(* IEC 61131-3 sources: elnaProjects/ElpcLogic/PomarKc7Changed/FunctionBlocks, 112 files *)

(* ---- AOAlg.st ---- *)
FUNCTION_BLOCK AOAlg

VAR_IN_OUT
	StrAlg : struct_Alg;
END_VAR

VAR
	kran6Open : struct_PhaseAlgoritm;
	kran4Close : struct_PhaseAlgoritm;
	kran3bOpen : struct_PhaseAlgoritm;
	mvOff : struct_PhaseAlgoritm;
	kran1Close : struct_PhaseAlgoritm;
	kran2Close : struct_PhaseAlgoritm;
	kran3Close : struct_PhaseAlgoritm;
	kran5Open : struct_PhaseAlgoritm;
	autoPnsOff : struct_PhaseAlgoritm;
	pnsOn : struct_PhaseAlgoritm;
	Pg_VhodLessThen300 : struct_PhaseAlgoritm;
	Pg_VyhodLessThen300 : struct_PhaseAlgoritm;
	nu1off : struct_PhaseAlgoritm;
	nu2off : struct_PhaseAlgoritm;
	AutoNU_Off : struct_PhaseAlgoritm;
	timer600 : struct_PhaseAlgoritm;
	pnsOff : struct_PhaseAlgoritm;
	Avom1Off : struct_PhaseAlgoritm;
	Avom2Off : struct_PhaseAlgoritm;
	Avom3Off : struct_PhaseAlgoritm;
	Avom4Off : struct_PhaseAlgoritm;
	autoAVOMOff : struct_PhaseAlgoritm;
	timer5 : struct_PhaseAlgoritm;
	klapan1 : struct_PhaseAlgoritm;
	klapan2 : struct_PhaseAlgoritm;
	nu_On : struct_PhaseAlgoritm;
	Start_AO_From : struct_PhaseAlgoritm;
	fb_kran6Open : fb_ph_Kran;
	fb_pnsOn : fb_ph_Switch;
	fb_kran4Close : fb_ph_Kran;
	fb_kran3bOpen : fb_ph_Kran;
	fb_mvOff : fb_ph_SectionSwitch;
	fb_kran1Close : fb_ph_Kran;
	fb_kran2Close : fb_ph_Kran;
	fb_kran3Close : fb_ph_Kran;
	fb_kran5Open : fb_ph_Kran;
	fb_autoPnsOff : fb_ph_algoritm;
	fb_Pg_VhodLessThen300 : fb_ph_CustomPhase;
	fb_Pg_VyhodLessThen300 : fb_ph_CustomPhase;
	fb_nu1Off : fb_ph_OilPump;
	fb_nu2Off : fb_ph_OilPump;
	fb_autoNuOff : fb_ph_algoritm;
	fb_timer600 : fb_ph_Timer;
	fb_pnsOff : fb_ph_Switch;
	fb_Avom1Off : fb_ph_Switch;
	fb_Avom2Off : fb_ph_Switch;
	fb_Avom3Off : fb_ph_Switch;
	fb_Avom4Off : fb_ph_Switch;
	fb_autoAVOMOff : fb_ph_algoritm;
	fb_timer5 : fb_ph_Timer;
	fb_klapan1 : fb_ph_CustomPhase;
	fb_klapan2 : fb_ph_CustomPhase;
	fb_nu_On : fb_ph_CustomPhase;
	fb_Start_AO_From : fb_ph_CustomPhase;
	_sunpackerCommand : fb_sunpackerCommand;
	_statusAi : TYPE_StatusAi;
	_Answers : TYPE_Answers;
	_statusDualInput : TYPE_statusDualInput;
	_commandDualInput : TYPE_commandDualInput;
	_DualStateImAction : TYPE_DualStateImAction;
	_PhaseAlgoritmAction : TYPE_PhaseAlgoritmAction;
	source : BYTE;
	cmd : BYTE;
	lastCmd : BYTE;
	source_for_Status : BYTE;
	cmd_for_Status : BYTE;
	command_error_for_Status : BYTE;
	resetCmdTimer : TON;
	resetCmdTimerPriznak : BOOL;
	onInit : BOOL;
	waitReset : TON;
END_VAR

VAR_EXTERNAL
	IM : ImConfig;
	algoritms : AlgoritmsConfig;
	ai : AiConfig;
	protections : ProtectionsConfig;
	ModeGpa : TYPE_ModeGpa;
	algManager : struct_AlgoritmsManager;
	AlgTimers : struct_AlgTimers;
END_VAR

VAR CONSTANT
	Ust_Pgaza : LREAL          := 0.3;
END_VAR

IF NOT onInit THEN
    fb_kran6Open(phaseNumber:=1, act:=_on);
    fb_kran4Close(phaseNumber:=2, act:=_off);
    fb_kran3bOpen(phaseNumber:=3, act:=_off);
    fb_mvOff(phaseNumber:=4, act:=_off);
    fb_kran1Close(phaseNumber:=5, act:=_off);
    fb_kran2Close(phaseNumber:=6, act:=_off);
    fb_kran3Close(phaseNumber:=7, act:=_off);
    fb_kran5Open(phaseNumber:=8, act:=_on);
    fb_autoPnsOff(phaseNumber:=9, act:=_reset, waitCompletion:=FALSE);
    fb_pnsOn(phaseNumber:=10, act:=_on);
    fb_Pg_VhodLessThen300(phaseNumber:=11);
    fb_Pg_VyhodLessThen300(phaseNumber:=12);
    fb_nu1Off(phaseNumber:=13, act:=_off);
    fb_nu2Off(phaseNumber:=14, act:=_off);
    fb_autoNuOff(phaseNumber:=15, act:=_reset, waitCompletion:=FALSE);
    fb_timer600(phaseNumber:=16, delay:=T#600S);
    fb_pnsOff(phaseNumber:=17, act:=_off);
    fb_Avom1Off(phaseNumber:=18, act:=_off);
    fb_Avom2Off(phaseNumber:=19, act:=_off);
    fb_Avom3Off(phaseNumber:=20, act:=_off);
    fb_Avom4Off(phaseNumber:=21, act:=_off);
    fb_autoAVOMOff(phaseNumber:=22, act:=_reset, waitCompletion:=FALSE);
    fb_timer5(phaseNumber:=23, delay:=T#5S);
    fb_klapan1(phaseNumber:=24);
    fb_klapan2(phaseNumber:=25);
    fb_nu_On(phaseNumber:=26);
    fb_Start_AO_From(phaseNumber:=27);
onInit:=TRUE;
END_IF;

fb_kran6Open(StrPh:=kran6Open, Im:=Im.kran6);
fb_pnsOn(StrPh:=pnsOn, Im:=Im.pns);
fb_kran4Close(StrPh:=kran4Close, Im:=Im.kran4);
fb_kran3bOpen(StrPh:=kran3bOpen, Im:=Im.kran3b);
fb_mvOff(StrPh:=mvOff, Im:=Im.mv);
fb_kran1Close(StrPh:=kran1Close, Im:=Im.kran1);
fb_kran2Close(StrPh:=kran2Close, Im:=Im.Kran2);
fb_kran3Close(StrPh:=kran3Close, Im:=Im.Kran3);
fb_kran5Open(StrPh:=kran5Open, Im:=Im.Kran5);
fb_autoPnsOff(StrPh:=autoPnsOff, alg:=algoritms.autoPns);
fb_Pg_VhodLessThen300(StrPh:=Pg_VhodLessThen300);
fb_Pg_VyhodLessThen300(StrPh:=Pg_VyhodLessThen300);
fb_nu1Off(StrPh:=nu1off, Im:=Im.nu1);
fb_nu2Off(StrPh:=nu2off, Im:=Im.nu2);
fb_autoNuOff(StrPh:=AutoNU_Off, alg:=algoritms.autoNu);
fb_timer600(StrPh:=timer600, timer:=AlgTimers.No_wait600);
fb_pnsOff(StrPh:=pnsOff, Im:=Im.pns);
fb_Avom1Off(StrPh:=Avom1Off, Im:=Im.v1_Avom);
fb_Avom2Off(StrPh:=Avom2Off, Im:=Im.v2_Avom);
fb_Avom3Off(StrPh:=Avom3Off, Im:=Im.v3_Avom);
fb_Avom4Off(StrPh:=Avom4Off, Im:=Im.v4_Avom);
fb_autoAVOMOff(StrPh:=autoAVOMOff, alg:=algoritms.AutoAvom);
fb_timer5(StrPh:=timer5, timer:=AlgTimers.No_wait5);
fb_klapan1(StrPh:=klapan1);
fb_klapan2(StrPh:=klapan2);
fb_nu_On(StrPh:=nu_On);
fb_Start_AO_From(StrPh:=Start_AO_From);

StrAlg.CanRun := StrAlg.inCanRun;
StrAlg.OpcCommandsDisabled := StrAlg.inOpcCommandsDisabled;

IF StrAlg.isRuning THEN

    IF	(*algoritms.F3.Smazka_1_2 OR*) IM.kran1.onStatus = _statusDualInput.STATUS_ON OR IM.kran1.onStatus = _statusDualInput.STATUS_TRANSITIONAL
	    OR IM.kran2.onStatus = _statusDualInput.STATUS_ON OR IM.kran2.onStatus = _statusDualInput.STATUS_TRANSITIONAL  THEN
	    IF (*(algoritms.F3.Smazka_1_2 OR*) IM.kran1.onStatus = _statusDualInput.STATUS_ON OR IM.kran1.onStatus = _statusDualInput.STATUS_TRANSITIONAL AND NOT klapan1.start AND NOT kran1Close.top THEN
		    runPhase(klapan1);
	    END_IF;
	    IF (*algoritms.F3.Smazka_1_2 OR*) IM.kran2.onStatus = _statusDualInput.STATUS_ON OR IM.kran2.onStatus = _statusDualInput.STATUS_TRANSITIONAL AND NOT klapan2.start AND NOT kran2Close.top THEN
		    runPhase(klapan2);
    	END_IF;
	(*algoritms.F3.Smazka_1_2:=FALSE; у меня нет такой штуки*)
    END_IF;

   (* IF NOT kran6Open.start THEN
	    ystavki.Block_kr6_alg.setValue (1);
	    IF IM.kran6._cmdreset.IN = FALSE THEN
		    ystavki.Block_kr6_alg.setValue (0); такой штуки тоже нет
		        runPhase(kran6Open);
	    END_IF;
    END_IF;*)

    (*IF NOT kran4Close.start THEN
	    ystavki.Block_kr4_alg.setValue (1);
	    IF IM.kran4._cmdreset.IN = FALSE THEN
		    ystavki.Block_kr4_alg.setValue (0);
		    kran4Close.run();
	    END_IF;
    END_IF;*)

    (*IF NOT kran3bOpen.start THEN
	    ystavki.Block_kr3b_alg.setValue (1);
	    IF IM.kran3b._cmdreset.IN = FALSE THEN
		    ystavki.Block_kr3b_alg.setValue (0);
		    runPhase(kran3bOpen);
	    END_IF;
    END_IF;*)

    resetDiProtection(protections.mvOff);
    resetDiProtection(protections.Off_avar_vikluchatel);
    resetDiProtection(protections.Reg_vozb_off);
    resetDiProtection(protections.Kran1_sdvig);
    resetDiProtection(protections.Kran2_sdvig);
    runPhase(mvOff);

    (*IF NOT kran1Close.start THEN
	ystavki.Block_kr1_alg.setValue (1);*)
	    (*IF IM.kran1._cmdreset.IN = FALSE THEN
		    ystavki.Block_kr1_alg.setValue (0);
		    runPhase(kran1Close);
	    END_IF;
    END_IF;*)

    (*IF NOT kran2Close.start THEN
	    ystavki.Block_kr2_alg.setValue (1);
	    IF IM.kran2._cmdreset.IN = FALSE THEN
		    ystavki.Block_kr2_alg.setValue (0);
		    runPhase(kran2Close);
	    END_IF;
    END_IF;*)

    (*IF NOT kran3Close.start THEN
	    ystavki.Block_kr3_alg.setValue (1);
	    IF	IM.kran3._cmdreset.IN = FALSE THEN
		    ystavki.Block_kr3_alg.setValue (0);
		    runPhase(kran3Close);
	    END_IF;
    END_IF;*)

    (*IF kran6Open.top THEN
	    algoritms.S_Vibr.CanRun:=FALSE;
	    algoritms.S_Vibr.reset ();
    END_IF;*)

    IF klapan1.start AND kran1Close.top THEN
	    (*IM.Kr1_Smazka.impulse();*)
	    klapan1.top:=TRUE;
    END_IF;
    IF	klapan2.start AND kran2Close.top THEN
	    (*zIM.Kr2_Smazka.impulse();*)
	    klapan2.top:=TRUE;
    END_IF;

    (*IF 	kran1Close.top AND kran2Close.top AND kran3Close.top AND kran4Close.top AND NOT kran5Open.top THEN
	    IF	NOT	kran5Open.start THEN
            ystavki.Block_kr5_alg.setValue (1);
		    IF	IM.kran5._cmdreset.IN = FALSE THEN
			    ystavki.Block_kr5_alg.setValue (0);
			    runPhase(kran5Open);
		    END_IF;
	    END_IF;

	    resetAiProtection(protections.Pgaza_na_vyhode_nagnetatelia);
    END_IF; *)

    IF mvOff.top (*AND NOT flag1*) THEN
	    (*algoritms.AutoPNS_Start.canrun :=FALSE;
	    algoritms.AutoPNS_Start.reset ();*)
	    algoritms.autoPns.canrun :=FALSE;
	    runPhase(autoPnsOff);
	    runPhase(pnsOn);
	    runPhase(nu_On);
	    (*vkluchit nasosi*)
	    algoritms.autoNu.canrun:=FALSE;
	    (*algoritms.autoNu_2.reset ();
	    algoritms.autoNu_1.canrun:=TRUE;
	    algoritms.autoNu_1.run ();
	    flag1:=TRUE;*)
    END_IF;

    IF	IM.nu1.onStatus =_statusDualInput.STATUS_ON OR IM.nu2.onStatus =_statusDualInput.STATUS_ON AND nu_On.start AND NOT nu_On.top THEN
	    nu_On.top:=TRUE;
    END_IF;

    IF kran5Open.top THEN
	    runPhase(Pg_VhodLessThen300);
	    runPhase(Pg_VyhodLessThen300);
	END_IF;

    IF Pg_VhodLessThen300.start AND NOT Pg_VhodLessThen300.top THEN
	    IF ai.Pgaza_na_vhode_nagnetatelia.interval >= _statusAi.NORMAL AND ai.Pgaza_na_vhode_nagnetatelia.value < 0.3 THEN
		    Pg_VhodLessThen300.top:=TRUE;
	    END_IF;
    END_IF;

    IF Pg_VyhodLessThen300.start AND NOT Pg_VyhodLessThen300.top THEN
	    IF ai.Pgaza_na_vyhode_nagnetatelia.interval>=_statusAi.NORMAL AND ai.Pgaza_na_vyhode_nagnetatelia.value < 0.3 THEN
		    Pg_VyhodLessThen300.top:=TRUE;
	    END_IF;
    END_IF;

    IF Pg_VhodLessThen300.top AND Pg_VyhodLessThen300.top AND pnsOn.top AND nu_On.top AND mvOff.top THEN
	    runPhase(nu1Off);
    	    resetAiProtection(protections.dPmaslo_gaz);
	    resetDiProtection(protections.dPmaslo_gaz_less100);
	    runAiProtection(protections.Pgaza_na_vhode_nagnetatelia_GPA_STOP);
	    runAiProtection(protections.Pgaza_na_vyhode_nagnetatelia_GPA_STOP);
	    AutoNU_Off.top:=TRUE;
    	(*algoritms.autoNu_1.CanRun:=FALSE;
	    algoritms.autoNu_1.reset ();*)
    END_IF;

    (*IF nuOff.top THEN
	    IF NOT algmanager.reg_V AND NOT pnsoff.start THEN
		    runPhase(timer600);
	    END_IF;
	    IF	NOT pnsoff.start THEN
		    sbrosVibeg.ask();
	    END_IF;
    END_IF;*)

    IF timer600.top (*OR sbrosVibeg.answer=Answers.ANS_YES*)  THEN
	    runPhase(pnsOff);
	    resetAiProtection(protections.Pmaslo_sm_nizkoe);
	    resetAiProtection(protections.Pmaslo_sm_vysokoe);
	    (*resetPhase(sbrosVibeg);*)
	    resetPhase(timer600);
	    (*algoritms.F2_Ch.autoAVOM_canrun_flag:=FALSE;
	    algoritms.F2_R.autoAVOM_canrun_flag:=FALSE;*)
    END_IF;

    IF (*NOT algoritms.F2_Ch.autoAVOM_canrun_flag AND NOT algoritms.F2_R.autoAVOM_canrun_flag AND*) pnsoff.start THEN
	    runPhase(Avom1Off);
	    runPhase(Avom2Off);
	    runPhase(Avom3Off);
	    runPhase(Avom4Off);
	    (*algoritms.R_AutoAVOM.CanRun:=FALSE;
	    algoritms.R_AutoAVOM.reset();
	    algoritms.S_AutoAVOM.CanRun:=FALSE;
	    algoritms.S_AutoAVOM.reset();
	    algoritms.Auto_Avom_.CanRun:=FALSE;*)
	    runPhase(autoAVOMOff);
    END_IF;

    IF pnsOff.top AND Avom1Off.top AND Avom2Off.top AND Avom3Off.top AND Avom4Off.top AND autoAVOMOff.top  THEN
	    runPhase(timer5);
    END_IF;

    IF timer5.top THEN
	    runPhase(timer5);
    END_IF;
END_IF;

_sunpackerCommand(command := StrAlg.inCommand);
	source := _sunpackerCommand.source;
	cmd := _sunpackerCommand.cmd;

IF cmd <> 0 AND lastCmd <> cmd AND (((NOT StrAlg.opcCommandsDisabled) AND source > 0) OR source = 0) then
	CASE BYTE_TO_INT(cmd) OF
		(*cmdRun*) 1: 	IF (StrAlg.CanRun) THEN
					StrAlg.isRuning := TRUE;
					StrAlg.isEnded := FALSE;
					StrAlg.hasError := FALSE;
					(*****************       OnRun       *****************)

                                                  algManager.nMode:=ModeGpa.MODE_NO;
                                                  (*runIfNotRunningSO(IM.SingleOutputs.Lampa_NO);*)

                                                  runPhase(kran4Close);
                                                  (*runPhase(timer120);*)
                                                  runPhase(nu1Off);
                                                  runPhase(timer600);

                                                 (* resetAiProtection(protections.Pgaza_na_vyhode_nagnetatelia);
                                                  resetAiProtection(protections.dPmaslo_gaz);
                                                  resetAiProtection(protections.Pmaslo_sm_nizkoe);
                                                  resetAiProtection(protections.Pmaslo_sm_vysokoe);
                                                  resetAiProtection(protections.Pgaza_na_vhode_nagnetatelia);
                                                  resetAiProtection(protections.Pgaza_na_vyhode_nagnetatelia);
                                                  resetDiProtection(protections.Reg_vozb_off);
                                                  resetDiProtection(protections.Fail_chastotnii_pusk);*)

					cmd_for_Status := cmd;
					source_for_Status := source;
					command_error_for_Status := 0;
				ELSE
					StrAlg.isRuning := FALSE;
					StrAlg.isEnded := FALSE;
					StrAlg.hasError 	:= FALSE;

					cmd_for_Status := 0;
					source_for_Status := source;
					command_error_for_Status := cmd;
				END_IF;
		(*cmdReset*) 2: 	StrAlg.isRuning := FALSE;
				StrAlg.isEnded := FALSE;
				StrAlg.hasError 	:= FALSE;

                                         (*****************       OnReset       *****************)
                                        waitReset(IN:=FALSE);
                                        (*resetIfRunningSO(IM.SingleOutputs.Lampa_NO);*)
                                        resetIfRunning(algoritms.vibegPNS);
                                        (*impulseSO(Im.SingleOutputs.SbrosBREO);*)

                                        (*resetPhase(timer120);*)
                                        resetPhase(kran6Open);
                                        resetPhase(pnsOn);
                                        resetPhase(kran4Close);
                                        resetPhase(kran3bOpen);
                                        resetPhase(mvOff);
                                        resetPhase(kran1Close);
                                        resetPhase(kran2Close);
                                        resetPhase(kran3Close);
                                        resetPhase(kran5Open);
	                              (*resetPhase(error_Krans);*)
                                        resetPhase(autoPnsOff);
                                        resetPhase(pnsOn);
                                        resetPhase(Pg_VhodLessThen300);
                                        resetPhase(Pg_VyhodLessThen300);
                                        resetPhase(nu2Off);
                                        resetPhase(nu1Off);
                                        resetPhase(AutoNU_Off);
                                        resetPhase(timer600);

				cmd_for_Status := cmd;
				source_for_Status := source;
				command_error_for_Status := 0;
	END_CASE;
	resetCmdTimer(IN := false);
	resetCmdTimerPriznak := TRUE;
END_IF;
lastCmd := cmd;

resetCmdTimer(IN := resetCmdTimerPriznak, PT := T#5S);
IF resetCmdTimer.Q THEN
	resetCmdTimerPriznak := FALSE;
	source_for_Status := 0;
	cmd_for_Status := 0;
	command_error_for_Status := 0;
END_IF;

StrAlg.Start:= kran6Open.startStatus
            OR pnsOn.startStatus
            OR kran4Close.startStatus
            OR kran3bOpen.startStatus
            OR mvOff.startStatus
            OR kran1Close.startStatus
            OR kran2Close.startStatus
            OR kran3Close.startStatus
            OR kran5Open.startStatus
            OR Pg_VhodLessThen300.startStatus
            OR nu1off.startStatus
            OR nu2off.startStatus
            OR Pg_VyhodLessThen300.startStatus
            OR AutoNU_Off.startStatus
            OR timer600.startStatus
            OR pnsOff.startStatus
            OR Avom1Off.startStatus
            OR Avom2Off.startStatus
            OR Avom3Off.startStatus
            OR Avom4Off.startStatus
            OR autoAVOMOff.startStatus
            OR timer5.startStatus
            OR klapan1.startStatus
            OR klapan2.startStatus
            OR nu_On.startStatus
            OR Start_AO_From.startStatus;

StrAlg.Error:= kran6Open.errorStatus
            OR pnsOn.errorStatus
            OR kran4Close.errorStatus
            OR kran3bOpen.errorStatus
            OR mvOff.errorStatus
            OR kran1Close.errorStatus
            OR kran2Close.errorStatus
            OR kran3Close.errorStatus
            OR kran5Open.errorStatus
            OR Pg_VhodLessThen300.errorStatus
            OR nu1off.errorStatus
            OR nu2off.errorStatus
            OR Pg_VyhodLessThen300.errorStatus
            OR AutoNU_Off.errorStatus
            OR timer600.errorStatus
            OR pnsOff.errorStatus
            OR Avom1Off.errorStatus
            OR Avom2Off.errorStatus
            OR Avom3Off.errorStatus
            OR Avom4Off.errorStatus
            OR autoAVOMOff.errorStatus
            OR timer5.errorStatus
            OR klapan1.errorStatus
            OR klapan2.errorStatus
            OR nu_On.errorStatus
            OR Start_AO_From.errorStatus;

StrAlg.Top:= kran6Open.topStatus
            OR pnsOn.topStatus
            OR kran4Close.topStatus
            OR kran3bOpen.topStatus
            OR mvOff.topStatus
            OR kran1Close.topStatus
            OR kran2Close.topStatus
            OR kran3Close.topStatus
            OR kran5Open.topStatus
            OR Pg_VhodLessThen300.topStatus
            OR nu1off.topStatus
            OR nu2off.topStatus
            OR Pg_VyhodLessThen300.topStatus
            OR AutoNU_Off.topStatus
            OR timer600.topStatus
            OR pnsOff.topStatus
            OR Avom1Off.topStatus
            OR Avom2Off.topStatus
            OR Avom3Off.topStatus
            OR Avom4Off.topStatus
            OR autoAVOMOff.topStatus
            OR timer5.topStatus
            OR klapan1.topStatus
            OR klapan2.topStatus
            OR nu_On.topStatus
            OR Start_AO_From.topStatus;

(*TODO: TYPE PROGRAM CODE HERE*)
StrAlg.status :=  SHL(BYTE_TO_DWORD(source_for_Status), 29)
			OR SHL(BYTE_TO_DWORD(cmd_for_Status), 26)
			OR SHL(BYTE_TO_DWORD(command_error_for_Status), 23)
			OR SHL(BOOL_TO_DWORD(StrAlg.OpcCommandsDisabled ), 21)
			OR SHL(BOOL_TO_DWORD(StrAlg.hasError),4)
			OR SHL(BOOL_TO_DWORD(StrAlg.CanRun),2)
			OR SHL(BOOL_TO_DWORD(StrAlg.isEnded),1)
			OR BOOL_TO_DWORD(StrAlg.isRuning);

(* ---- ApuskAlg.st ---- *)
FUNCTION_BLOCK ApuskAlg

VAR_IN_OUT
	StrAlg : struct_Alg;
END_VAR

VAR
	runOilsystem : struct_PhaseAlgoritm;
	runEngine : struct_PhaseAlgoritm;
	filling : struct_PhaseAlgoritm;
	fb_runOilsystem : fb_ph_algoritm;
	fb_runEngine : fb_ph_algoritm;
	fb_filling : fb_ph_algoritm;
	_sunpackerCommand : fb_sunpackerCommand;
	_PhaseAlgoritmAction : TYPE_PhaseAlgoritmAction;
	_statusDualInput : TYPE_statusDualInput;
	source : BYTE;
	cmd : BYTE;
	lastCmd : BYTE;
	source_for_Status : BYTE;
	cmd_for_Status : BYTE;
	command_error_for_Status : BYTE;
	resetCmdTimer : TON;
	resetCmdTimerPriznak : BOOL;
	onInit : BOOL;
	waitReset : TON;
END_VAR

VAR_EXTERNAL
	algoritms : AlgoritmsConfig;
	ModeGpa : TYPE_ModeGpa;
	algManager : struct_AlgoritmsManager;
	IM : ImConfig;
END_VAR

IF NOT onInit THEN

         fb_runOilsystem(phaseNumber:=0, act:=_run, waitCompletion:=TRUE);
            fb_runEngine(phaseNumber:=1, act:=_run, waitCompletion:=TRUE);
              fb_filling(phaseNumber:=2, act:=_run, waitCompletion:=TRUE);

onInit:=TRUE;
END_IF;

         fb_runOilsystem(StrPh:=runOilsystem, alg:=algoritms.puskOilSystem);
            fb_runEngine(StrPh:=runEngine, alg:=algoritms.engineRun);
              fb_filling(StrPh:=filling, alg:=algoritms.filling);

StrAlg.CanRun := StrAlg.inCanRun;
StrAlg.OpcCommandsDisabled := StrAlg.inOpcCommandsDisabled;

IF StrAlg.isRuning THEN

    StrAlg.hasError := runOilsystem.error OR runEngine.error OR filling.error;

    IF runOilsystem.top THEN
         runPhase(runEngine);
    END_IF;

    IF runEngine.top THEN
         runPhase(filling);
    END_IF;

    IF filling.top THEN
          waitReset(IN:=TRUE, PT:= T#2S);
    END_IF;

    IF waitReset.Q THEN

        IF Im.kran6.onStatus = _statusDualInput.STATUS_On THEN
	algManager.nMode:= ModeGpa.MODE_WORK_Ring;
        END_IF;
        IF Im.kran6.onStatus = _statusDualInput.STATUS_Off THEN
	algManager.nMode:= ModeGpa.MODE_WORK_Line;
        END_IF;

        resetIfRunning(StrAlg);
    END_IF;

    StrAlg.isEnded:= filling.top;

END_IF;

StrAlg.CanRun := StrAlg.inCanRun;
StrAlg.OpcCommandsDisabled := StrAlg.inOpcCommandsDisabled;

(* ---- Если управление с ВУ заблокировано, то  передаем команду из алгоритма ---- *)
IF StrAlg.inOpcCommandsDisabled THEN
	StrAlg.inCommand := StrAlg.inCommand_Alg;
ELSE (* иначе передаем команду с АРМа*)
	StrAlg.inCommand := StrAlg.inCommand_ARM;
END_IF;

_sunpackerCommand(command := StrAlg.inCommand);
	source := _sunpackerCommand.source;
	cmd := _sunpackerCommand.cmd;

IF cmd <> 0 AND lastCmd <> cmd AND (((NOT StrAlg.opcCommandsDisabled) AND source > 0) OR source = 0) then
	CASE BYTE_TO_INT(cmd) OF
		(*cmdRun*) 1: 	IF (StrAlg.CanRun) THEN
					StrAlg.isRuning := TRUE;
					StrAlg.isEnded := FALSE;
					StrAlg.hasError := FALSE;
					(*****************       OnRun       *****************)

                                                  algoritms.puskOilSystem.inCanRun:= TRUE	;
                                                  algoritms.filling.inCanRun:= TRUE	;
                                                  algoritms.engineRun.inCanRun:= TRUE	;

                                                  algManager.nMode:=ModeGpa.MODE_APUSK;
                                                  (*impulseSO(Im.SingleOutputs.VzvodBREO);*)
                                                  runPhase(runOilsystem);

					cmd_for_Status := cmd;
					source_for_Status := source;
					command_error_for_Status := 0;
				ELSE
					StrAlg.isRuning := FALSE;
					StrAlg.isEnded := FALSE;
					StrAlg.hasError 	:= FALSE;

					cmd_for_Status := 0;
					source_for_Status := source;
					command_error_for_Status := cmd;
				END_IF;
		(*cmdReset*) 2: 	StrAlg.isRuning := FALSE;
				StrAlg.isEnded := FALSE;
				StrAlg.hasError 	:= FALSE;

                                         (*****************       OnReset       *****************)
                                        waitReset(IN:=FALSE);
                                        StrAlg.inCanRun:=FALSE;

                                        resetPhase(runOilsystem);
                                        resetPhase(runEngine);
                                        resetPhase(filling);

                                        StrAlg.inOpcCommandsDisabled:=FALSE;

				cmd_for_Status := cmd;
				source_for_Status := source;
				command_error_for_Status := 0;
	END_CASE;
	resetCmdTimer(IN := false);
	resetCmdTimerPriznak := TRUE;
END_IF;
lastCmd := cmd;

resetCmdTimer(IN := resetCmdTimerPriznak, PT := T#5S);
IF resetCmdTimer.Q THEN
	resetCmdTimerPriznak := FALSE;
	source_for_Status := 0;
	cmd_for_Status := 0;
	command_error_for_Status := 0;
END_IF;

StrAlg.Start:= runOilsystem.startStatus
            OR runEngine.startStatus
            OR filling.startStatus;

StrAlg.Error:= runOilsystem.errorStatus
            OR runEngine.errorStatus
            OR filling.errorStatus;

StrAlg.Top:=   runOilsystem.topStatus
            OR runEngine.topStatus
            OR filling.topStatus;

(*TODO: TYPE PROGRAM CODE HERE*)
StrAlg.status :=  SHL(BYTE_TO_DWORD(source_for_Status), 29)
			OR SHL(BYTE_TO_DWORD(cmd_for_Status), 26)
			OR SHL(BYTE_TO_DWORD(command_error_for_Status), 23)
			OR SHL(BOOL_TO_DWORD(StrAlg.OpcCommandsDisabled ), 21)
			OR SHL(BOOL_TO_DWORD(StrAlg.hasError),4)
			OR SHL(BOOL_TO_DWORD(StrAlg.CanRun),2)
			OR SHL(BOOL_TO_DWORD(StrAlg.isEnded),1)
			OR BOOL_TO_DWORD(StrAlg.isRuning);

(* ---- engineRunAlg.st ---- *)
FUNCTION_BLOCK engineRunAlg

VAR_IN_OUT
	StrAlg : struct_Alg;
END_VAR

VAR
	BreakPuskTimer : struct_PhaseAlgoritm;
	RunProtection_mvoff : struct_PhaseAlgoritm;
	LowOil_upStopust : struct_PhaseAlgoritm;
	mvOn : struct_PhaseAlgoritm;
	AutoPns_ph : struct_PhaseAlgoritm;
	AutoAvom_ph : struct_PhaseAlgoritm;
	pnsOff : struct_PhaseAlgoritm;
	testUnsuccessful : struct_PhaseAlgoritm;
	fb_BreakPuskTimer : fb_ph_Timer;
	fb_RunProtection_mvoff : fb_ph_DIprotection;
	fb_LowOil_upStopust : fb_ph_WaitAnalogValue;
	fb_mvOn : fb_ph_SectionSwitch;
	fb_AutoPns_ph : fb_ph_algoritm;
	fb_AutoAvom_ph : fb_ph_algoritm;
	fb_pnsOff : fb_ph_Switch;
	fb_testUnsuccessful : fb_ph_CustomPhase;
	_sunpackerCommand : fb_sunpackerCommand;
	_DualStateImAction : TYPE_DualStateImAction;
	_PhaseAlgoritmAction : TYPE_PhaseAlgoritmAction;
	source : BYTE;
	cmd : BYTE;
	lastCmd : BYTE;
	source_for_Status : BYTE;
	cmd_for_Status : BYTE;
	command_error_for_Status : BYTE;
	resetCmdTimer : TON;
	resetCmdTimerPriznak : BOOL;
	onInit : BOOL;
	waitReset : TON;
END_VAR

VAR_EXTERNAL
	IM : ImConfig;
	algoritms : AlgoritmsConfig;
	ai : AiConfig;
	protections : ProtectionsConfig;
	AlgTimers : struct_AlgTimers;
END_VAR

IF NOT onInit THEN

     fb_BreakPuskTimer(phaseNumber:=0, delay:=T#665S);
   fb_LowOil_upStopust(phaseNumber:=1);
               fb_mvOn(phaseNumber:=2, act:=_on);
         fb_AutoPns_ph(phaseNumber:=3, act:=_run, waitCompletion:=FALSE);
        fb_AutoAvom_ph(phaseNumber:=4, act:=_run, waitCompletion:=FALSE);
             fb_pnsOff(phaseNumber:=5, act:=_off);
fb_RunProtection_mvoff(phaseNumber:=7, act:=_run);
   fb_testUnsuccessful(phaseNumber:=17);

onInit:=TRUE;
END_IF;

        fb_BreakPuskTimer(StrPh:=BreakPuskTimer, timer:=AlgTimers.engineRun_BreakPuskTimer);
     (* fb_LowOil_upStopust(StrPh:=LowOil_upStopust, ai:=ai.Pmasla_posle_GNS, more:=im.AutoPns_UstStop.Value);*)
                  fb_mvOn(StrPh:=mvOn, Im:=Im.mv);
            fb_AutoPns_ph(StrPh:=AutoPns_ph, alg:=algoritms.AutoPns);
           fb_AutoAvom_ph(StrPh:=AutoAvom_ph, alg:=algoritms.AutoAvom);
                fb_pnsOff(StrPh:=pnsOff, Im:=Im.pns);
  (*fb_RunProtection_mvoff(StrPh:=RunProtection_mvoff, StrDiP:=protections.Pgaza_na_vyhode_nagnetatelia_GPA_STOP);*)
      fb_testUnsuccessful(StrPh:=testUnsuccessful);

StrAlg.CanRun := StrAlg.inCanRun;
StrAlg.OpcCommandsDisabled := StrAlg.inOpcCommandsDisabled;

IF StrAlg.isRuning THEN

    StrAlg.hasError := mvOn.error OR pnsOff.error OR testUnsuccessful.error;

    IF mvOn.top THEN
        runPhase(RunProtection_mvoff);
        runPhase(AutoAvom_ph);
        runPhase(LowOil_upStopust);
    END_IF;
    (*
    IF AutoAvom_ph.top THEN
        algoritms.AutoAvom.inOpcCommandsDisabled:=FALSE;
    END_IF;
    *)
    IF LowOil_upStopust.top THEN
        runPhase(pnsOff);
    END_IF;

    IF pnsOff.top THEN
       runPhase(AutoPns_ph);
    END_IF;

    IF BreakPuskTimer.top AND NOT AutoPns_ph.top THEN
          testUnsuccessful.error:=TRUE;
    END_IF;

    IF AutoPns_ph.top THEN
          resetPhase(BreakPuskTimer);
	waitReset(IN:=TRUE, PT:= T#2S);
    END_IF;

    IF waitReset.Q AND NOT (algoritms.Apusk.isRuning OR algoritms.SemiAutoPusk.isRuning) THEN
	resetIfRunning(StrAlg);
    END_IF;

    StrAlg.isEnded:= AutoPns_ph.top;
END_IF;

StrAlg.CanRun := StrAlg.inCanRun;
StrAlg.OpcCommandsDisabled := StrAlg.inOpcCommandsDisabled;

(* ---- Если управление с ВУ заблокировано, то  передаем команду из алгоритма ---- *)
IF StrAlg.inOpcCommandsDisabled THEN
	StrAlg.inCommand := StrAlg.inCommand_Alg;
ELSE (* иначе передаем команду с АРМа*)
	StrAlg.inCommand := StrAlg.inCommand_ARM;
END_IF;

_sunpackerCommand(command := StrAlg.inCommand);
	source := _sunpackerCommand.source;
	cmd := _sunpackerCommand.cmd;

IF cmd <> 0 AND lastCmd <> cmd AND (((NOT StrAlg.opcCommandsDisabled) AND source > 0) OR source = 0) then
	CASE BYTE_TO_INT(cmd) OF
		(*cmdRun*) 1: 	IF (StrAlg.CanRun) THEN
					StrAlg.isRuning := TRUE;
					StrAlg.isEnded := FALSE;
					StrAlg.hasError := FALSE;
					(*****************       OnRun       *****************)

                                                  runPhase(mvOn);
                                                  runPhase(BreakPuskTimer);
                                                  runPhase(testUnsuccessful);

					cmd_for_Status := cmd;
					source_for_Status := source;
					command_error_for_Status := 0;
				ELSE
					StrAlg.isRuning := FALSE;
					StrAlg.isEnded := FALSE;
					StrAlg.hasError 	:= FALSE;

					cmd_for_Status := 0;
					source_for_Status := source;
					command_error_for_Status := cmd;
				END_IF;
		(*cmdReset*) 2: 	StrAlg.isRuning := FALSE;
				StrAlg.isEnded := FALSE;
				StrAlg.hasError 	:= FALSE;

                                         (*****************       OnReset       *****************)
                                        StrAlg.inCanRun:=FALSE;
                                        waitReset(IN:=FALSE);

                                        resetPhase(BreakPuskTimer);
                                        resetPhase(RunProtection_mvoff);
                                        resetPhase(LowOil_upStopust);
                                        resetPhase(mvOn);
                                        resetPhase(AutoPns_ph);
                                        resetPhase(AutoAvom_ph);
                                        resetPhase(pnsOff);
                                        resetPhase(testUnsuccessful);

				cmd_for_Status := cmd;
				source_for_Status := source;
				command_error_for_Status := 0;
	END_CASE;
	resetCmdTimer(IN := false);
	resetCmdTimerPriznak := TRUE;
END_IF;
lastCmd := cmd;

resetCmdTimer(IN := resetCmdTimerPriznak, PT := T#5S);
IF resetCmdTimer.Q THEN
	resetCmdTimerPriznak := FALSE;
	source_for_Status := 0;
	cmd_for_Status := 0;
	command_error_for_Status := 0;
END_IF;

StrAlg.Start:= BreakPuskTimer.startStatus
            OR RunProtection_mvoff.startStatus
            OR LowOil_upStopust.startStatus
            OR mvOn.startStatus
            OR AutoPns_ph.startStatus
            OR AutoAvom_ph.startStatus
            OR pnsOff.startStatus
            OR testUnsuccessful.startStatus;

StrAlg.Error:= BreakPuskTimer.errorStatus
            OR RunProtection_mvoff.errorStatus
            OR LowOil_upStopust.errorStatus
            OR mvOn.errorStatus
            OR AutoPns_ph.errorStatus
            OR AutoAvom_ph.errorStatus
            OR pnsOff.errorStatus
            OR testUnsuccessful.errorStatus;

StrAlg.Top:=   BreakPuskTimer.topStatus
            OR RunProtection_mvoff.topStatus
            OR LowOil_upStopust.topStatus
            OR mvOn.topStatus
            OR AutoPns_ph.topStatus
            OR AutoAvom_ph.topStatus
            OR pnsOff.topStatus
            OR testUnsuccessful.topStatus;

(*TODO: TYPE PROGRAM CODE HERE*)
StrAlg.status :=  SHL(BYTE_TO_DWORD(source_for_Status), 29)
			OR SHL(BYTE_TO_DWORD(cmd_for_Status), 26)
			OR SHL(BYTE_TO_DWORD(command_error_for_Status), 23)
			OR SHL(BOOL_TO_DWORD(StrAlg.OpcCommandsDisabled ), 21)
			OR SHL(BOOL_TO_DWORD(StrAlg.hasError),4)
			OR SHL(BOOL_TO_DWORD(StrAlg.CanRun),2)
			OR SHL(BOOL_TO_DWORD(StrAlg.isEnded),1)
			OR BOOL_TO_DWORD(StrAlg.isRuning);

(* ---- ExtNarabotka.st ---- *)
FUNCTION_BLOCK ExtNarabotka

VAR
	saveInterval : TIME          := T#30S;
	narabotka : UDINT;
	timer : RTC;
	saveTimer : TON;
END_VAR

VAR_IN_OUT
	retain_narabotka : UDINT;
END_VAR

VAR
	initialized : BOOL;
END_VAR

VAR_INPUT
	started : BOOL;
	reset : BOOL;
END_VAR

IF NOT initialized THEN
	narabotka:=retain_narabotka;
	initialized:=TRUE;
END_IF;

timer();

IF timer.Q THEN
	narabotka:=DT_TO_UDINT( timer.CDT);

END_IF;
saveTimer(IN:=TRUE, PT:=saveInterval);
IF saveTimer.Q THEN
	retain_narabotka:=narabotka;
	saveTimer(IN:=FALSE);
END_IF;

IF started THEN
	IF NOT timer.Q THEN
		timer.PDT:=UDINT_TO_DT(narabotka);
                    timer.IN:=TRUE;
	END_IF;
ELSE
	IF timer.Q THEN
		timer.IN:=FALSE;
                    saveTimer.IN:=FALSE;
	END_IF;
END_IF;

IF reset THEN
timer.PDT:=UINT_TO_DT(0);
IF timer.IN THEN
	timer(IN:=FALSE);
	timer(IN:=TRUE);
END_IF;
narabotka:=0;
reset:=FALSE;
END_IF;

(* ---- fb_AI_Init.st ---- *)
FUNCTION_BLOCK fb_AI_Init

VAR_INPUT
	data_Ini : BOOL; (*Флаг необходимости инициализации параметров.*)
	dLL : LREAL;
	dHL : LREAL;
	dLA : LREAL;
	dHA : LREAL;
	dLW : LREAL;
	dHW : LREAL;
	ISVALIDREF_LA : BOOL          := False;
	ISVALIDREF_HA : BOOL          := False;
	ISVALIDREF_LW : BOOL          := False;
	ISVALIDREF_HW : BOOL          := False;
	delayLA : TIME          := T#0S;
	delayLW : TIME          := T#0S;
	delayHW : TIME          := T#0S;
	delayHA : TIME          := T#0S;
	inpLL : LREAL          := 4000.0;
	inpHL : LREAL          := 20000.0;
	CurrentShotCircuit : LREAL          := 21000.0;
	CurrentBreakCircuit : LREAL          := 3700.0;
	dMaxChangeSpeed : LREAL;
	dMaxChangeSpeedDown : LREAL;
	histeresis : LREAL;
	aperturFilter : LREAL;
	exponentialFilter : LREAL;
	rassoglasovanie : LREAL;
	inOpcCommandsDisabled : BOOL;
END_VAR

VAR_IN_OUT
	strAI : struct_AI; (*Дескриптор AI-канала.*)
END_VAR

VAR_OUTPUT
	Init : BOOL          := FALSE; (*Флаг успешно выполненной инициализации.*)
END_VAR

(*****            Функциональный блок переинициализации структуры-дескриптора канала аналогового ввода.            *****)
     Init := false;

    IF data_Ini THEN                            (* Параметрам требуется переинициализация. *)
        strAI.dLL                := dLL;
        strAI.dHL                := dHL;
        strAI.dLA                := dLA;
        strAI.dHA                := dHA;
        strAI.dLW                := dLW;
        strAI.dHW                := dHW;
        strAI.ISVALIDREF_LA      := ISVALIDREF_LA;
        strAI.ISVALIDREF_HA      := ISVALIDREF_HA;
        strAI.ISVALIDREF_LW      := ISVALIDREF_LW;
        strAI.ISVALIDREF_HW      := ISVALIDREF_HW;
        strAI.delayLA            := delayLA;
        strAI.delayLW            := delayLW;
        strAI.delayHW            := delayHW;
        strAI.delayHA            := delayHA;
        strAI.inpLL              := inpLL;
        strAI.inpHL              := inpHL;
        strAI.CurrentShotCircuit := CurrentShotCircuit;
        strAI.CurrentBreakCircuit:= CurrentBreakCircuit;
        strAI.dMaxChangeSpeed     := dMaxChangeSpeed;
        strAI.dMaxChangeSpeedDown := dMaxChangeSpeedDown;
        strAI.histeresis         := histeresis;
        strAI.aperturFilter      := aperturFilter;
        strAI.exponentialFilter  := exponentialFilter;
        strAI.rassoglasovanie    := rassoglasovanie;
        strAI.rassoglasovanie    := rassoglasovanie;

        data_Ini:=false;
        Init := TRUE;
     END_IF;
  IF Init THEN
        dLL:= 0.0;
        dHL:= 0.0;
        dLA:= 0.0;
        dHA:= 0.0;
        dLW:= 0.0;
        dHW:= 0.0;
        inpLL:= 4000.0;
        inpHL:= 20000.0;
        CurrentShotCircuit:= 21000.0;
        CurrentBreakCircuit:= 3700.0;
        ISVALIDREF_LA:= false;
        ISVALIDREF_HA:= false;
        ISVALIDREF_LW:= false;
        ISVALIDREF_HW:= false;
        delayLA:= T#0S;
        delayLW:= T#0S;
        delayHW:= T#0S;
        delayHA:= T#0S;
        dMaxChangeSpeed:= 0.0;
        dMaxChangeSpeedDown:= 0.0;
        histeresis:= 0.0;
        aperturFilter:= 0.0;
        exponentialFilter:= 0.0;
        rassoglasovanie:= 0.0;
      END_IF;

(* ---- fb_AiProtection.st ---- *)
FUNCTION_BLOCK fb_AiProtection

VAR_INPUT
	ai : struct_AI;
END_VAR

VAR_IN_OUT
	StrAIp : struct_AiProtection;
END_VAR

VAR
	_sunpackerCommand : fb_sunpackerCommand;
	_signalingTp : TOF;
	_statusAi : TYPE_StatusAi;
	source : BYTE;
	cmd : BYTE;
	lastCmd : BYTE;
	source_for_Status : BYTE;
	cmd_for_Status : BYTE;
	command_error_for_Status : BYTE;
	resetCmdTimer : TON;
	resetCmdTimerPriznak : BOOL;
	signalinTimer : TON;
	timer : TON;
	SignalingTrig : R_TRIG;
	SignalingFTrig : F_TRIG;
	SignalingAi : BOOL;
END_VAR

timer(IN :=(ai.interval=StrAIp.controlLimit) AND (ai.interval >= _statusAi.normal) AND StrAIp.isRunning, PT :=StrAIp.delay);
SignalingTrig(CLK := timer.Q);
IF SignalingTrig.Q THEN
	SignalingAi := TRUE;
END_IF;
SignalingFTrig(CLK := timer.Q);
IF SignalingFTrig.Q THEN
	SignalingAi := FALSE;
END_IF;

StrAIp.Tag := StrAIp.inTag;
StrAIp.RunOnStart := StrAIp.inRunOnStart;

StrAIp.CanRun := StrAIp.inCanRun;

StrAIp.OpcCommandsDisabled := StrAIp.inOpcCommandsDisabled;

(* ---- Если управление с ВУ заблокировано, то передаем команду из алгоритма ---- *)
IF StrAIp.inOpcCommandsDisabled THEN
	StrAIp.inCommand := StrAIp.inCommand_Alg;
ELSE (* иначе передаем команду с АРМа*)
	StrAIp.inCommand := StrAIp.inCommand_ARM;
END_IF;

_sunpackerCommand(command := StrAIp.inCommand);
	source := _sunpackerCommand.source;
	cmd := _sunpackerCommand.cmd;

IF cmd <> 0 AND lastCmd <> cmd AND (((NOT StrAIp.opcCommandsDisabled) AND source > 0) OR source = 0) then

	CASE BYTE_TO_INT(cmd) OF
		(*cmdRun*) 1: 	IF        NOT StrAIp.Remont THEN
					StrAIp.isEnded := FALSE;
					StrAIp.hasError 	:= FALSE;
					StrAIp.isRunning := TRUE;

					cmd_for_Status := cmd;
					source_for_Status := source;
					command_error_for_Status := 0;
				ELSE
					StrAIp.isRunning := FALSE;
					StrAIp.isEnded := FALSE;
					StrAIp.hasError 	:= FALSE;

					cmd_for_Status := 0;
					source_for_Status := source;
					command_error_for_Status := cmd;
				END_IF;
                                        StrAIp.inopcCommandsDisabled:=FALSE;

		(*cmdReset*) 2: 	StrAIp.isRunning := FALSE;
				StrAIp.isEnded := FALSE;
				StrAIp.hasError 	:= FALSE;
				SignalingAi := FALSE;
				StrAIp.Check := FALSE;
                                        (*StrAIp.Remont := FALSE;*)
				cmd_for_Status := cmd;
				source_for_Status := source;
				command_error_for_Status := 0;
                                        StrAIp.inopcCommandsDisabled:=FALSE;

	(*cmd_setRemont*) 4 :	StrAIp.Remont := TRUE;
				(*StrAIp.isRunning := FALSE;*)

				cmd_for_Status := cmd;
				source_for_Status := source;
				command_error_for_Status := 0;
	(*cmd_resetRemont*) 5 : 	(*IF (ai.interval=StrAIp.controlLimit) THEN
					cmd_for_Status := 0;
					source_for_Status := 0;
					command_error_for_Status := cmd;
				ELSE*)
					StrAIp.Remont := FALSE;
					(*StrAIp.isRunning := TRUE;*)

					cmd_for_Status := cmd;
					source_for_Status := source;
					command_error_for_Status := 0;
				(*END_IF;*)
	(*cmd_setCheck*) 6 : 	StrAIp.Check := TRUE;

				cmd_for_Status := cmd;
				source_for_Status := source;
				command_error_for_Status := 0;
	END_CASE;
	resetCmdTimer(IN := false);
	resetCmdTimerPriznak := TRUE;
END_IF;
lastCmd := cmd;

resetCmdTimer(IN := resetCmdTimerPriznak);
IF resetCmdTimer.Q THEN
	resetCmdTimerPriznak := FALSE;
	source_for_Status := 0;
	cmd_for_Status := 0;
	command_error_for_Status := 0;
END_IF;

IF StrAIp.isRunning AND NOT StrAIp.Remont AND NOT StrAIp.Check THEN
	StrAIp.Signaling := SignalingAi;
	StrAIp.SignalingTP := _signalingTp.Q;
ELSE
	StrAIp.Signaling := 0;
	StrAIp.SignalingTP := 0;
END_IF;

_signalingTp(in := StrAIp.Signaling, PT := T#1s);

StrAIp.status :=  SHL(BYTE_TO_DWORD(source_for_Status), 29)
			OR SHL(BYTE_TO_DWORD(cmd_for_Status), 26)
			OR SHL(BYTE_TO_DWORD(command_error_for_Status), 23)
			OR SHL(BOOL_TO_DWORD(StrAIp.OpcCommandsDisabled ), 21)
			OR SHL(BOOL_TO_DWORD(StrAIp.Signaling), 16)
			OR SHL(BOOL_TO_DWORD(StrAIp.RunOnStart ), 15)
			OR SHL(BOOL_TO_DWORD(StrAIp.remont), 6)
			OR SHL(BOOL_TO_DWORD(StrAIp.Check), 5)
			OR SHL(BOOL_TO_DWORD(StrAIp.hasError), 4)
			OR SHL(BOOL_TO_DWORD(StrAIp.SignalingTP), 3)
			OR SHL(BOOL_TO_DWORD(StrAIp.CanRun), 2)
			OR SHL(BOOL_TO_DWORD(StrAIp.isEnded), 1)
			OR BOOL_TO_DWORD(StrAIp.isRunning);

(* ---- fb_AiProtection_Init.st ---- *)
FUNCTION_BLOCK fb_AiProtection_Init

VAR_INPUT
	data_Ini : BOOL; (*Флаг необходимости инициализации параметров.*)
	controlLimit : BYTE;
	delay : TIME;
	inTag : BYTE;
	inRunOnStart : BOOL;
END_VAR

VAR_IN_OUT
	str_AIp : struct_AiProtection;
END_VAR

VAR_OUTPUT
	Init : BOOL          := FALSE; (*Флаг успешно выполненной инициализации.*)
END_VAR

(*****            Функциональный блок переинициализации структуры  AiProtection          *****)

 Init := FALSE;

    IF data_Ini THEN                            (* Параметрам требуется переинициализация. *)
        str_AIp.controlLimit        := controlLimit;
        str_AIp.delay               := delay;
        str_AIp.inTag               := inTag;
        str_AIp.inRunOnStart        := inRunOnStart;

        data_Ini:=FALSE;
        Init := TRUE;
    END_IF;
    IF Init THEN
        controlLimit:= 0;
        delay:= T#0S;
        inTag:= 0;
        inRunOnStart:= FALSE;
    END_IF;

(* ---- fb_AiSourceMlp.st ---- *)
FUNCTION_BLOCK fb_AiSourceMlp

VAR_INPUT
	arAIN : TItemAIN; (*Данные от модуля AI*)
	err_mod : TItemDIN; (*Диагностика от модуля AI*)
END_VAR

VAR_IN_OUT
	strAI : struct_AI; (*Текущие параметры канала AI*)
END_VAR

VAR
	_statusAi : TYPE_StatusAi;
	_commandAnalog : TYPE_CommandAnalog;
	_sunpackerCommand : fb_sunpackerCommand;
	_AnalogLimitFlags : TYPE_AnalogLimitFlags;
	notReliable : BOOL;
	_lastValue : LREAL;
	resetCmdTimer : TON;
	_LastValueTimer : TON;
	resetCmdTimerPriznak : BOOL;
	k : LREAL;
	b : LREAL;
	ap : LREAL;
	raznitsa : LREAL;
	rABS : LREAL;
	h : LREAL;
	mismatch : LREAL;
	parametr : BYTE;
	source : BYTE;
	cmd : BYTE;
	lastCmd : BYTE;
	source_for_Status : BYTE;
	cmd_for_Status : BYTE;
	command_error_for_Status : BYTE;
	onInit : BOOL;
	off_trig : R_TRIG;
	on_trig : R_TRIG;
	remont_trig : R_TRIG;
	LL_trig : R_TRIG;
	HL_trig : R_TRIG;
	Normal_trig : R_TRIG;
	Nedostover_trig : R_TRIG;
END_VAR

strAI.opcCommandsDisabled := strAI.inopcCommandsDisabled ;

(* ---- При первом пуске принимаем значение уставок ---- *)
IF NOT onInit THEN

          strAI.LL := strAI.dLL;
          strAI.HL := strAI.dHL;

          strAI.MaxChangeSpeed     := strAI.dMaxChangeSpeed;
          strAI.MaxChangeSpeedDown := strAI.dMaxChangeSpeedDown;

          IF strAI.ISVALIDREF_HA THEN strAI.HA := strAI.dHA; END_IF;

          IF strAI.ISVALIDREF_LA THEN strAI.LA := strAI.dLA; END_IF;

          IF strAI.ISVALIDREF_HW THEN strAI.HW := strAI.dHW; END_IF;

          IF strAI.ISVALIDREF_LW THEN strAI.LW := strAI.dLW; END_IF;

	onInit  := TRUE;
END_IF;

(* ---- пересчет тока в физ величину ---- *)
k := (strAI.HL - strAI.LL)/(strAI.inpHl - strAI.inpLL);
b := strAI.LL - k * strAI.inpLL;
strAI.value := k * arAIN.dblValue + b;

(* ---- определение обрыва и кз ----- *)

strAI.blConnect :=(*(UINT_TO_WORD(arAIN.wFlags) = 1472) and*) (UINT_TO_WORD(err_mod.wValue) = 20) and (UINT_TO_WORD(err_mod.wFlags) = 192);
IF NOT strAI.blConnect THEN
    strAI.interval := _statusAi.NOTDEFINED;
ELSIF ((arAIN.dblValue < strAI.currentBreakCircuit) AND (strAI.currentBreakCircuit > 0.0)) OR ((strAI.interval = _statusAi.LL) AND (arAIN.dblValue < (strAI.currentBreakCircuit + 100.0))) THEN
    strAI.interval := _statusAi.LL;
ELSIF ((arAIN.dblValue > strAI.currentShotCircuit) AND (strAI.currentShotCircuit > 0.0)) OR ((strAI.interval = _statusAi.HL) AND (arAIN.dblValue > (strAI.currentShotCircuit - 100.0))) THEN
    strAI.interval := _statusAi.HL;
ELSE
    strAI.interval := _statusAi.normal;
END_IF;

IF NOT strAI.imit THEN
	(* Расчет апертурного фильтра*)
	ap := strAI.aperturFilter * 0.01 * (strAI.HL - strAI.LL);
	IF strAI.aperturFilter <> 0.0 THEN raznitsa := strAI.value- _lastValue;
		IF 	raznitsa < 0.0 	THEN 	rABS := -raznitsa; 		ELSE 	rABS := raznitsa; 		END_IF;
		IF 	rABS > ap 	THEN 	strAI.value := strAI.value;	ELSE 	strAI.value := _lastValue; 	END_IF;
	END_IF;

	(* Расчет экпоненциального фильтра*)
	IF strAI.exponentialFilter <> 0.0 THEN strAI.value := (strAI.exponentialFilter * strAI.value) + ((1.0 - strAI.exponentialFilter) * _lastValue); END_IF;
ELSE
	strAI.interval := _statusAi.normal;
END_IF;

IF notReliable THEN strAI.interval := _statusAi.NOTRELIABLE; END_IF;

IF NOT notReliable THEN
	IF strAI.interval >= _statusAi.normal THEN
		strAI.interval := _statusAi.NOTDEFINED;
		h := strAI.histeresis* 0.01 * (strAI.HL-strAI.LL);
		(*определение выхода за аппаратные границы вынесено в GetData.здесь только для нужд имитации*)
		IF strAI.imit THEN
			mismatch := strAI.rassoglasovanie * 0.01 * (strAI.HL - strAI.LL);
			IF ( strAI.value < strAI.LL - mismatch)   THEN strAI.interval := _statusAi.LL;
			ELSIF  (strAI.value > strAI.Hl + mismatch) THEN strAI.interval := _statusAi.HL; END_IF;
		ELSE
			strAI.interval := _statusAi.normal;
			IF strAI.ISVALIDREF_LA AND NOT strAI.Disabled_LA AND (strAI.interval = _statusAi.normal) THEN
				IF (strAI.value  < strAI.LA) OR ((strAI.interval = _statusAi.LA)  AND ((strAI.value - h) < strAI.LA))  THEN
					strAI.interval := _statusAi.LA;
				END_IF;
			END_IF;
			IF strAI.ISVALIDREF_HA  AND NOT strAI.Disabled_HA AND (strAI.interval = _statusAi.normal)  THEN
				IF (strAI.value > strAI.HA) OR ((strAI.interval = _statusAi.HA)  AND ((strAI.value + h) > strAI.HA))  THEN
					strAI.interval := _statusAi.HA;
				END_IF;
			END_IF;
			IF strAI.ISVALIDREF_LW AND NOT strAI.Disabled_LW AND (strAI.interval = _statusAi.normal)  THEN
				IF (strAI.value < strAI.LW) OR ((strAI.interval = _statusAi.LW)  AND ((strAI.value - h) < strAI.LW)) THEN
					strAI.interval := _statusAi.LW;
				END_IF;
			END_IF;
			IF strAI.ISVALIDREF_HW AND NOT strAI.Disabled_HW  AND (strAI.interval = _statusAi.normal) THEN
				IF (strAI.value > strAI.HW)  OR ((strAI.interval = _statusAi.HW)  AND ((strAI.value + h) > strAI.HW))   THEN
					strAI.interval := _statusAi.HW;
				END_IF;
			END_IF;
		END_IF;
	END_IF;
ELSE
	strAI.interval := _statusAi.NOTRELIABLE;
END_IF;

IF strAI.remont THEN strAI.interval := _statusAi.NOTDEFINED; END_IF;

(* ---- Если управление с ВУ заблокировано, то  передаем команду из алгоритма ---- *)
IF strAI.inOpcCommandsDisabled THEN
	strAI.inCommand := strAI.inCommand_Alg;
ELSE (* иначе передаем команду с АРМа*)
	strAI.inCommand := strAI.inCommand_ARM;
END_IF;

_sunpackerCommand(command := strAI.inCommand);
	source := _sunpackerCommand.source;
	parametr := _sunpackerCommand.parametr;
	cmd := _sunpackerCommand.cmd;

IF cmd <> 0 AND lastCmd <> cmd and (((NOT strAI.opcCommandsDisabled) AND source > 0) OR source = 0) then
	CASE BYTE_TO_INT(cmd) OF
	(*cmd_SetUstavki*) 1 :
				IF ((parametr AND _AnalogLimitFlags.LL) <> 0)		             	THEN 	strAI.LL := strAI.dLL; END_IF;
				IF ((parametr AND _AnalogLimitFlags.HL) <> 0)		 	          THEN	strAI.HL := strAI.dHL; END_IF;
				IF ((parametr AND _AnalogLimitFlags.LA) <> 0) AND strAI.ISVALIDREF_LA 	THEN	strAI.LA := strAI.dLA; END_IF;
				IF ((parametr AND _AnalogLimitFlags.HA) <> 0) AND strAI.ISVALIDREF_HA 	THEN	strAI.HA := strAI.dHA; END_IF;
				IF ((parametr AND _AnalogLimitFlags.LW) <> 0) AND strAI.ISVALIDREF_LW 	THEN	strAI.LW := strAI.dLW; END_IF;
				IF ((parametr AND _AnalogLimitFlags.HW) <> 0) AND strAI.ISVALIDREF_HW 	THEN	strAI.HW := strAI.dHW; END_IF;
                                        IF ((parametr AND _AnalogLimitFlags.SipUP) <> 0)                       	THEN	strAI.MaxChangeSpeed     := strAI.dMaxChangeSpeed;     END_IF;
				IF ((parametr AND _AnalogLimitFlags.SipDown) <> 0)                      	THEN	strAI.MaxChangeSpeedDown := strAI.dMaxChangeSpeedDown; END_IF;

	(*cmd_SetRemont*) 6 :
				strAI.remont := TRUE;
	(*cmd_ResetRemont*) 7 :
				strAI.remont := FALSE;
	(*cmd_kvitNotReliable*) 4 :
				notReliable := FALSE;
	END_CASE;
	source_for_Status := source;
	cmd_for_Status := cmd;
	command_error_for_Status := 0;
	resetCmdTimer(IN := FALSE);
	resetCmdTimerPriznak := TRUE;
END_IF;
lastCmd := cmd;

resetCmdTimer(IN := resetCmdTimerPriznak, PT := T#5S);
IF resetCmdTimer.Q THEN
	resetCmdTimerPriznak := FALSE;
	source_for_Status := 0;
	cmd_for_Status := 0;
	command_error_for_Status := 0;
END_IF;

strAI.NS_Min := (strAI.value < strAI.minValue) AND strAI.minValue_ISVALIDREF;
strAI.NS_Max := (strAI.value > strAI.maxValue) AND strAI.maxValue_ISVALIDREF;

strAI.NS := (strAI.interval <= _statusAi.normal) AND NOT strAI.remont;

Normal_trig(CLK := strAI.interval >= _statusAi.normal);

IF NOT Normal_trig.Q THEN
	_LastValueTimer(PT := T#1S);
	IF (strAI.value<>_lastValue) OR _LastValueTimer.Q THEN
		IF (_LastValueTimer.ET>T#0MS) THEN
			strAI.ChangeSpeed:=(strAI.value-_lastValue)/(TIME_TO_LREAL(_LastValueTimer.ET));
		END_IF;
		_LastValueTimer(IN:=FALSE);

		_LastValueTimer(IN:=TRUE);
	END_IF;
END_IF;
_lastValue := strAI.value;

IF ((strAI.maxChangeSpeed<>0.0) OR  (strAI.maxChangeSpeedDown<>0.0)) AND ( strAI.interval>=_statusAi.normal) THEN
		IF (strAI.ChangeSpeed>0.0) THEN
		    IF (strAI.ChangeSpeed > strAI.maxChangeSpeed) AND (strAI.maxChangeSpeed>0.0000001) THEN
			 notReliable:=TRUE;
		    END_IF;
		ELSE
		    IF (ABS(strAI.ChangeSpeed)>strAI.maxChangeSpeedDown) AND (strAI.maxChangeSpeedDown>0.0000001)  THEN
                               notReliable:=TRUE;
		    END_IF;
		END_IF;

END_IF;

strAI.status := SHL(BYTE_TO_DWORD(source_for_Status), 29) 		              (* Источник команды *)
			OR SHL(BYTE_TO_DWORD(cmd_for_Status), 26) 	    (* Команда *)
			OR SHL(BYTE_TO_DWORD(command_error_for_Status), 23)   (* Ошибка команды *)
			OR SHL(BOOL_TO_DWORD(strAI.OpcCommandsDisabled ), 21) (* Управление в ВУ заблокировано *)
			OR SHL(BOOL_TO_DWORD(strAI.Disabled_HA), 9)		    (* ВА исключена из формирования интервала *)
			OR SHL(BOOL_TO_DWORD(strAI.Disabled_LA), 8)		    (* НА исключена из формирования интервала *)
			OR SHL(BOOL_TO_DWORD(strAI.Disabled_HW), 7)		    (* ВП исключена из формирования интервала *)
			OR SHL(BOOL_TO_DWORD(strAI.Disabled_LW), 6)	              (* НП исключена из формирования интервала *)
			OR SHL(BOOL_TO_DWORD(strAI.NS), 5)			    (* неиспарвность сигнала *)
			OR SHL(BOOL_TO_DWORD(strAI.remont), 4)	              (* Выведен в ремонт *)
			OR BYTE_TO_DWORD(strAI.interval);	              (* интервал *)

(* ---- fb_AiSourceMlp_timer.st ---- *)
FUNCTION_BLOCK fb_AiSourceMlp_timer

VAR_INPUT
	arAIN : TItemAIN; (*Данные от модуля AI*)
	err_mod : TItemDIN; (*Диагностика от модуля AI*)
END_VAR

VAR_IN_OUT
	strAI : struct_AI; (*Текущие параметры канала AI*)
END_VAR

VAR
	_statusAi : TYPE_StatusAi;
	_commandAnalog : TYPE_CommandAnalog;
	_sunpackerCommand : fb_sunpackerCommand;
	_AnalogLimitFlags : TYPE_AnalogLimitFlags;
	notReliable : BOOL;
	_lastValue : LREAL;
	resetCmdTimer : TON;
	_LastValueTimer : TON;
	resetCmdTimerPriznak : BOOL;
	k : LREAL;
	b : LREAL;
	ap : LREAL;
	raznitsa : LREAL;
	rABS : LREAL;
	h : LREAL;
	mismatch : LREAL;
	parametr : BYTE;
	source : BYTE;
	cmd : BYTE;
	lastCmd : BYTE;
	source_for_Status : BYTE;
	cmd_for_Status : BYTE;
	command_error_for_Status : BYTE;
	secondTakt : BOOL;
	off_trig : R_TRIG;
	on_trig : R_TRIG;
	remont_trig : R_TRIG;
	LL_trig : R_TRIG;
	HL_trig : R_TRIG;
	Normal_trig : R_TRIG;
	Nedostover_trig : R_TRIG;
	timerLA : TON;
	timerHA : TON;
	timerLW : TON;
	timerHW : TON;
END_VAR

VAR RETAIN
	retainLL : LREAL; (*Текущее значение ВГ*)
	retainHL : LREAL; (*Текущее значение НГ*)
	retainLA : LREAL; (*Текущее значение НА*)
	retainHA : LREAL; (*Текущее значение ВА*)
	retainLW : LREAL; (*Текущее значение НП*)
	retainHW : LREAL; (*Текущее значение ВП*)
END_VAR

strAI.opcCommandsDisabled := strAI.inopcCommandsDisabled ;

(* ---- При первом пуске принимаем значение уставок ---- *)
IF NOT secondTakt THEN
          IF (strAI.dLL <> retainLL) AND (retainLL <> 0.0) THEN  strAI.LL := retainLL;
          ELSE strAI.LL := strAI.dLL; END_IF;
	IF (strAI.dHL <> retainHL) AND (retainHL <> 0.0) THEN  strAI.HL := retainHL;
          ELSE strAI.HL := strAI.dHL; END_IF;

          IF strAI.ISVALIDREF_HA AND (strAI.dHA <> retainHA) AND (retainHA <> 0.0) THEN  strAI.HA := retainHA;
          ELSE strAI.HA := strAI.dHA; END_IF;

          IF strAI.ISVALIDREF_LA AND (strAI.dLA <> retainLA) AND (retainLA <> 0.0) THEN  strAI.LA := retainLA;
          ELSE strAI.LA := strAI.dLA; END_IF;

          IF strAI.ISVALIDREF_HW AND (strAI.dHW <> retainHW) AND (retainHW <> 0.0) THEN  strAI.HW := retainHW;
          ELSE strAI.HW := strAI.dHW; END_IF;

          IF strAI.ISVALIDREF_LW AND (strAI.dLW <> retainLW) AND (retainLW <> 0.0) THEN  strAI.LW := retainLW;
          ELSE strAI.LW := strAI.dLW; END_IF;

	secondTakt  := TRUE;
END_IF;

(* ---- пересчет тока в физ величину ---- *)
k := (strAI.HL - strAI.LL)/(strAI.inpHl - strAI.inpLL);
b := strAI.LL - k * strAI.inpLL;
strAI.value := k * arAIN.dblValue + b;

(* ---- определение обрыва и кз ----- *)

strAI.blConnect := true;(*(UINT_TO_WORD(arAIN.wFlags) = 1472) and (UINT_TO_WORD(err_mod.wValue) = 20) and (UINT_TO_WORD(err_mod.wFlags) = 192); *)
IF NOT strAI.blConnect THEN
    strAI.interval := _statusAi.NOTDEFINED;
ELSIF ((arAIN.dblValue < strAI.currentBreakCircuit) AND (strAI.currentBreakCircuit > 0.0)) OR ((strAI.interval = _statusAi.LL) AND (arAIN.dblValue < (strAI.currentBreakCircuit + 100.0))) THEN
    strAI.interval := _statusAi.LL;
ELSIF ((arAIN.dblValue > strAI.currentShotCircuit) AND (strAI.currentShotCircuit > 0.0)) OR ((strAI.interval = _statusAi.HL) AND (arAIN.dblValue > (strAI.currentShotCircuit - 100.0))) THEN
    strAI.interval := _statusAi.HL;
ELSE
    strAI.interval := _statusAi.normal;
END_IF;

IF NOT strAI.imit THEN
	(* Расчет апертурного фильтра*)
	ap := strAI.aperturFilter * 0.01 * (strAI.HL - strAI.LL);
	IF strAI.aperturFilter <> 0.0 THEN raznitsa := strAI.value- _lastValue;
		IF 	raznitsa < 0.0 	THEN 	rABS := -raznitsa; 		ELSE 	rABS := raznitsa; 		END_IF;
		IF 	rABS > ap 	THEN 	strAI.value := strAI.value;	ELSE 	strAI.value := _lastValue; 	END_IF;
	END_IF;

	(* Расчет экпоненциального фильтра*)
	IF strAI.exponentialFilter <> 0.0 THEN strAI.value := (strAI.exponentialFilter * strAI.value) + ((1.0 - strAI.exponentialFilter) * _lastValue); END_IF;
ELSE
	strAI.interval := _statusAi.normal;
END_IF;

IF notReliable THEN strAI.interval := _statusAi.NOTRELIABLE; END_IF;

IF NOT notReliable THEN
	IF strAI.interval >= _statusAi.normal THEN
		strAI.interval := _statusAi.NOTDEFINED;
		h := strAI.histeresis* 0.01 * (strAI.HL-strAI.LL);
		(*определение выхода за аппаратные границы вынесено в GetData.здесь только для нужд имитации*)
		IF strAI.imit THEN
			mismatch := strAI.rassoglasovanie * 0.01 * (strAI.HL - strAI.LL);
			IF ( strAI.value < strAI.LL - mismatch)   THEN strAI.interval := _statusAi.LL;
			ELSIF  (strAI.value > strAI.Hl + mismatch) THEN strAI.interval := _statusAi.HL; END_IF;
		ELSE
			strAI.interval := _statusAi.normal;
			IF strAI.ISVALIDREF_LA AND NOT strAI.Disabled_LA AND (strAI.interval = _statusAi.normal) THEN
                              timerLA(IN:=(strAI.value  < strAI.LA) OR ((strAI.interval = _statusAi.LA)  AND ((strAI.value - h) < strAI.LA)), PT:=strAI.delayLA);
				IF timerLA.Q  THEN
					strAI.interval := _statusAi.LA;
				END_IF;
			END_IF;
			IF strAI.ISVALIDREF_HA  AND NOT strAI.Disabled_HA AND (strAI.interval = _statusAi.normal)  THEN
                              timerHA(IN:=(strAI.value > strAI.HA) OR ((strAI.interval = _statusAi.HA)  AND ((strAI.value + h) > strAI.HA)), PT:=strAI.delayHA);
				IF timerHA.Q  THEN
					strAI.interval := _statusAi.HA;
				END_IF;
			END_IF;
			IF strAI.ISVALIDREF_LW AND NOT strAI.Disabled_LW AND (strAI.interval = _statusAi.normal)  THEN
                              timerLW(IN:=(strAI.value < strAI.LW) OR ((strAI.interval = _statusAi.LW)  AND ((strAI.value - h) < strAI.LW)), PT:=strAI.delayLW);
				IF timerLW.Q THEN
					strAI.interval := _statusAi.LW;
				END_IF;
			END_IF;
			IF strAI.ISVALIDREF_HW AND NOT strAI.Disabled_HW  AND (strAI.interval = _statusAi.normal) THEN
                              timerHW(IN:=(strAI.value > strAI.HW)  OR ((strAI.interval = _statusAi.HW)  AND ((strAI.value + h) > strAI.HW)), PT:=strAI.delayHW);
				IF  timerHW.Q  THEN
					strAI.interval := _statusAi.HW;
				END_IF;
			END_IF;
		END_IF;
	END_IF;
ELSE
	strAI.interval := _statusAi.NOTRELIABLE;
END_IF;

IF strAI.remont THEN strAI.interval := _statusAi.NOTDEFINED; END_IF;

_sunpackerCommand(command := strAI.inCommand);
	source := _sunpackerCommand.source;
	parametr := _sunpackerCommand.parametr;
	cmd := _sunpackerCommand.cmd;

IF cmd <> 0 AND lastCmd <> cmd and (((NOT strAI.opcCommandsDisabled) AND source > 0) OR source = 0) then
	CASE BYTE_TO_INT(cmd) OF
	(*cmd_SetUstavki*) 1 :
				IF ((parametr AND _AnalogLimitFlags.LL) <> 0)		             	THEN 	strAI.LL := strAI.dLL; retainLL:= strAI.LL; END_IF;
				IF ((parametr AND _AnalogLimitFlags.HL) <> 0)		 	          THEN	strAI.HL := strAI.dHL; retainHL:= strAI.HL; END_IF;
				IF ((parametr AND _AnalogLimitFlags.LA) <> 0) AND strAI.ISVALIDREF_LA 	THEN	strAI.LA := strAI.dLA; retainLA:= strAI.LA; END_IF;
				IF ((parametr AND _AnalogLimitFlags.HA) <> 0) AND strAI.ISVALIDREF_HA 	THEN	strAI.HA := strAI.dHA; retainHA:= strAI.HA; END_IF;
				IF ((parametr AND _AnalogLimitFlags.LW) <> 0) AND strAI.ISVALIDREF_LW 	THEN	strAI.LW := strAI.dLW; retainLW:= strAI.LW; END_IF;
				IF ((parametr AND _AnalogLimitFlags.HW) <> 0) AND strAI.ISVALIDREF_HW 	THEN	strAI.HW := strAI.dHW; retainHW:= strAI.HW; END_IF;
	(*cmd_SetRemont*) 2 :
				strAI.remont := TRUE;
	(*cmd_ResetRemont*) 3 :
				strAI.remont := FALSE;
	(*cmd_kvitNotReliable*) 4 :
				notReliable := FALSE;
	END_CASE;
	source_for_Status := source;
	cmd_for_Status := cmd;
	command_error_for_Status := 0;
	resetCmdTimer(IN := FALSE);
	resetCmdTimerPriznak := TRUE;
END_IF;
lastCmd := cmd;

resetCmdTimer(IN := resetCmdTimerPriznak, PT := T#5S);
IF resetCmdTimer.Q THEN
	resetCmdTimerPriznak := FALSE;
	source_for_Status := 0;
	cmd_for_Status := 0;
	command_error_for_Status := 0;
END_IF;

strAI.NS_Min := (strAI.value < strAI.minValue) AND strAI.minValue_ISVALIDREF;
strAI.NS_Max := (strAI.value > strAI.maxValue) AND strAI.maxValue_ISVALIDREF;

strAI.NS := (strAI.interval <= _statusAi.normal) AND NOT strAI.remont;

Normal_trig(CLK := strAI.interval >= _statusAi.normal);

IF NOT Normal_trig.Q THEN
	_LastValueTimer(PT := T#1S);
	IF (strAI.value<>_lastValue) OR _LastValueTimer.Q THEN
		IF (_LastValueTimer.ET>T#0MS) THEN
			strAI.ChangeSpeed:=(strAI.value-_lastValue)/(TIME_TO_LREAL(_LastValueTimer.ET)/1000.0);
		END_IF;
		_LastValueTimer(IN:=FALSE);

		_LastValueTimer(IN:=TRUE);
	END_IF;
END_IF;
_lastValue := strAI.value;

IF ((strAI.maxChangeSpeed<>0.0) OR  (strAI.maxChangeSpeedDown<>0.0)) AND ( strAI.interval>=_statusAi.normal) THEN
		IF (strAI.ChangeSpeed>0.0) THEN
		    IF (strAI.ChangeSpeed > strAI.maxChangeSpeed) AND (strAI.maxChangeSpeed>0.0000001) THEN
			 notReliable:=TRUE;
		    END_IF;
		ELSE
		    IF (ABS(strAI.ChangeSpeed)>strAI.maxChangeSpeedDown) AND (strAI.maxChangeSpeedDown>0.0000001)  THEN
                               notReliable:=TRUE;
		    END_IF;
		END_IF;

END_IF;

strAI.status := SHL(BYTE_TO_DWORD(source_for_Status), 29) 		              (* Источник команды *)
			OR SHL(BYTE_TO_DWORD(cmd_for_Status), 26) 	    (* Команда *)
			OR SHL(BYTE_TO_DWORD(command_error_for_Status), 23)   (* Ошибка команды *)
			OR SHL(BOOL_TO_DWORD(strAI.OpcCommandsDisabled ), 21) (* Управление в ВУ заблокировано *)
			OR SHL(BOOL_TO_DWORD(strAI.Disabled_HA), 9)		    (* ВА исключена из формирования интервала *)
			OR SHL(BOOL_TO_DWORD(strAI.Disabled_LA), 8)		    (* НА исключена из формирования интервала *)
			OR SHL(BOOL_TO_DWORD(strAI.Disabled_HW), 7)		    (* ВП исключена из формирования интервала *)
			OR SHL(BOOL_TO_DWORD(strAI.Disabled_LW), 6)	              (* НП исключена из формирования интервала *)
			OR SHL(BOOL_TO_DWORD(strAI.NS), 5)			    (* неиспарвность сигнала *)
			OR SHL(BOOL_TO_DWORD(strAI.remont), 4)	              (* Выведен в ремонт *)
			OR BYTE_TO_DWORD(strAI.interval);	              (* интервал *)

(* ---- fb_AlgoritmsManager.st ---- *)
FUNCTION_BLOCK fb_AlgoritmsManager

VAR_IN_OUT
	str_AM : struct_AlgoritmsManager;
END_VAR

VAR
	onInit : BOOL;
END_VAR

VAR_EXTERNAL
	ai : AiConfig;
END_VAR

VAR
	EoTrig : R_TRIG;
	EoFTrig : F_TRIG;
	PsLampTrig : R_TRIG;
	PsLampFTrig : F_TRIG;
	Ring : R_TRIG;
	Line : R_TRIG;
	statusDualInput : TYPE_statusDualInput;
END_VAR

VAR_EXTERNAL
	IM : ImConfig;
	protections : ProtectionsConfig;
	algoritms : AlgoritmsConfig;
	ModeGpa : TYPE_ModeGpa;
END_VAR

IF NOT onInit THEN
          DisableAiLimits(ai);
          (*IM.SingleSignals.P_oil_low.Disabled_Sig:=TRUE;
          IM.SingleSignals.dP_oilgaz_low.Disabled_Sig:=TRUE;*)
          str_AM.nMode:=ModeGpa.MODE_STOP;
          BlockAllIM(IM);
          runIfNotRunning(algoritms.AutoTen);
onInit:=TRUE;
END_IF;

str_AM.DiscretPS:=anyDiscretPS(IM);
str_AM.AnalogsPs:=anyAnalogsPs(ai);
str_AM.ProtectionSignaling:=anyProtectionSignaling(protections);

(*EoTrig(CLK := IM.SingleSignals.BEO_Srabat.Q);*)
IF EoTrig.Q THEN
	stopPusk(algoritms);
	resetAndDisable(algoritms.Remont);
	resetAndDisable(algoritms.no);
	resetAndDisable(algoritms.ao);
	str_AM.nMode:=ModeGpa.MODE_EO;
END_IF;
(*EoFTrig(CLK := IM.SingleSignals.BEO_Srabat.Q);*)
IF EoFTrig.Q THEN
	str_AM.nMode:=ModeGpa.MODE_STOP;
	runIfNotRunning(algoritms.ao);
END_IF;

(*IF (str_AM.ProtectionSignaling OR Im.SingleSignals.AO_KC.Q OR Im.SingleSignals.AOGPA_knopkaSHU.Q OR Im.SingleSignals.AOGPA_PRU.Q )
	AND NOT((str_AM.mode=ModeGpa.MODE_AO) OR (str_AM.mode=ModeGpa.MODE_EO) OR IM.SingleOutputs.IndikicijaAS_fonar.Q
          OR (str_AM.mode=ModeGpa.MODE_TESTAZ) OR (str_AM.mode=ModeGpa.MODE_TESTDPMG) OR (str_AM.mode=ModeGpa.MODE_REMONT) OR
          (str_AM.mode=ModeGpa.MODE_TESTPMS))THEN
		runIfNotRunning(algoritms.ao);
	str_AM.nMode:=ModeGpa.MODE_AO;
END_IF;
*)
(*IF Im.SingleSignals.NOGPA_knopkaSHU.Q  AND algoritms.no.CanRun THEN
	runIfNotRunning(algoritms.no);
          str_AM.nMode:=ModeGpa.MODE_NO;
END_IF;*)

PsLampTrig(CLK := str_AM.DiscretPS OR str_AM.AnalogsPs);
(*IF PsLampTrig.Q THEN
          runIfNotRunningSO(IM.SingleOutputs.IndikicijaPS_fonar);
END_IF;*)
PsLampFTrig(CLK := str_AM.DiscretPS OR str_AM.AnalogsPs);
(*IF PsLampFTrig.Q THEN
          resetIfRunningSO(IM.SingleOutputs.IndikicijaPS_fonar);
END_IF;*)

IF str_AM.mode = ModeGpa.MODE_WORK_Line OR str_AM.mode = ModeGpa.MODE_WORK_Ring  THEN

	Ring(CLK:=Im.kran6.onStatus=statusDualInput.STATUS_On);
	Line(CLK:=Im.kran6.onStatus=statusDualInput.STATUS_Off);

	IF Ring.Q AND str_AM.mode = ModeGpa.MODE_WORK_Line THEN
		str_AM.nMode:=ModeGpa.MODE_WORK_Ring;
	END_IF;
	IF Line.Q AND str_AM.mode = ModeGpa.MODE_WORK_Ring THEN
		str_AM.nMode:=ModeGpa.MODE_WORK_Line;
	END_IF;

END_IF;

IF str_AM.mode = ModeGpa.MODE_WORK_Line THEN
          runIfNotRunning(alg:=algoritms.AntiPompag);
	ELSE
          resetAndDisable(alg:=algoritms.AntiPompag);
END_IF;

IF str_AM.nMode<>str_AM.mode THEN
	str_AM.mode:=str_AM.nMode;
	CASE str_AM.mode OF
	(*ModeGpa.MODE_REMONT*)1:
		stopPusk(algoritms);
		resetAndDisable(alg:=algoritms.no);
		resetAndDisable(alg:=algoritms.ao);
		resetAndDisable(alg:=algoritms.TestProtection);
                    resetAndDisable(alg:=algoritms.testIm);

	(*ModeGpa.MODE_TESTAZ*)16:
		stopPusk(algoritms);
		resetAndDisable(alg:=algoritms.ao);
		resetAndDisable(alg:=algoritms.no);
                    resetAndDisable(alg:=algoritms.Remont);
                    resetAndDisable(alg:=algoritms.testIm);

          (*ModeGpa.MODE_TESTIM*)15:
                    stopPusk(algoritms);
                    resetAndDisable(alg:=algoritms.Remont);
                    resetAndDisable(alg:=algoritms.TestProtection);

	(*ModeGpa.MODE_EO*)14:
		stopPusk(algoritms);
		resetAndDisable(alg:=algoritms.no);
		resetAndDisable(alg:=algoritms.ao);
		resetAndDisable(alg:=algoritms.Remont);
                    resetAndDisable(alg:=algoritms.testIm);
                    resetAndDisable(alg:=algoritms.TestProtection);
	(*ModeGpa.MODE_AO*)13:
		(*//stopPusk();*)
		resetAndDisable(alg:=algoritms.no);
		resetAndDisable(alg:=algoritms.Remont);
                    resetAndDisable(alg:=algoritms.testIm);
                    resetAndDisable(alg:=algoritms.TestProtection);
                    algoritms.VibegPNS.inCanRun:=TRUE;
	(*ModeGpa.MODE_NO*)12:
		stopPusk(algoritms);
                    resetAndDisable(alg:=algoritms.testIm);
                    resetAndDisable(alg:=algoritms.Remont);
                    resetAndDisable(alg:=algoritms.TestProtection);
                    algoritms.VibegPNS.inCanRun:=TRUE;
		algoritms.ao.inCanRun:=TRUE;
	(*ModeGpa.MODE_APUSK*)8:
		resetAndDisable(alg:=algoritms.SemiAutoPusk);
		resetAndDisable(alg:=algoritms.puskV);
		resetAndDisable(alg:=algoritms.puskK);
		resetAndDisable(alg:=algoritms.testdPmg);
		resetAndDisable(alg:=algoritms.testPms);
		(*resetAndDisable(alg:=algoritms.testIm);
                    resetAndDisable(alg:=algoritms.TestProtection);
                    resetAndDisable(alg:=algoritms.Remont);*)
		resetAndDisable(alg:=algoritms.ppu);
		algoritms.no.inCanRun:=TRUE;
		algoritms.ao.inCanRun:=TRUE;

	(*ModeGpa.MODE_MPUSK*)9:
		resetAndDisable(alg:=algoritms.Apusk);
		resetAndDisable(alg:=algoritms.puskV);
		resetAndDisable(alg:=algoritms.puskK);
		resetAndDisable(alg:=algoritms.testdPmg);
		resetAndDisable(alg:=algoritms.testPms);
		(*resetAndDisable(alg:=algoritms.testIm);
                    resetAndDisable(alg:=algoritms.TestProtection);
                    resetAndDisable(alg:=algoritms.Remont);	*)
		resetAndDisable(alg:=algoritms.ppu);
		algoritms.no.inCanRun:=TRUE;
                    algoritms.no.inOpcCommandsDisabled:=FALSE;
		algoritms.ao.inCanRun:=TRUE;
                    algoritms.ao.inOpcCommandsDisabled:=FALSE;

	(*ModeGpa.MODE_PUSKK*)5:
                    resetAndDisable(alg:=algoritms.ppu);
		resetAndDisable(alg:=algoritms.Apusk);
		resetAndDisable(alg:=algoritms.SemiAutoPusk);
		resetAndDisable(alg:=algoritms.TestProtection);
                    resetAndDisable(alg:=algoritms.Remont);
		resetAndDisable(alg:=algoritms.testIm	 );
		algoritms.no.inCanRun:=TRUE;
                    algoritms.no.inOpcCommandsDisabled:=FALSE;
		algoritms.ao.inCanRun:=TRUE;
                    algoritms.ao.inOpcCommandsDisabled:=FALSE;
	(*ModeGpa.MODE_PUSKV*)4:
                    resetAndDisable(alg:=algoritms.ppu);
		resetAndDisable(alg:=algoritms.Apusk);
		resetAndDisable(alg:=algoritms.SemiAutoPusk);
		resetAndDisable(alg:=algoritms.TestProtection);
                    resetAndDisable(alg:=algoritms.Remont);
		resetAndDisable(alg:=algoritms.testIm	 );
		algoritms.no.inCanRun:=TRUE;
                    algoritms.no.inOpcCommandsDisabled:=FALSE;
		algoritms.ao.inCanRun:=TRUE;
                    algoritms.ao.inOpcCommandsDisabled:=FALSE;

	(*ModeGpa.MODE_TESTDPMG*)6:
                    resetAndDisable(alg:=algoritms.ppu);
		resetAndDisable(alg:=algoritms.Apusk);
		resetAndDisable(alg:=algoritms.SemiAutoPusk);
		resetAndDisable(alg:=algoritms.TestProtection);
                    resetAndDisable(alg:=algoritms.Remont);
		resetAndDisable(alg:=algoritms.testIm	 );
		algoritms.no.inCanRun:=TRUE;
                    algoritms.no.inOpcCommandsDisabled:=FALSE;
		algoritms.ao.inCanRun:=TRUE;
                    algoritms.ao.inOpcCommandsDisabled:=FALSE;

	(*ModeGpa.MODE_TESTPMS*)7:
                    resetAndDisable(alg:=algoritms.ppu);
		resetAndDisable(alg:=algoritms.Apusk);
		resetAndDisable(alg:=algoritms.SemiAutoPusk);
		resetAndDisable(alg:=algoritms.TestProtection);
                    resetAndDisable(alg:=algoritms.Remont);
		resetAndDisable(alg:=algoritms.testIm);
		algoritms.no.inCanRun:=TRUE;
                    algoritms.no.inOpcCommandsDisabled:=FALSE;
		algoritms.ao.inCanRun:=TRUE;
                    algoritms.ao.inOpcCommandsDisabled:=FALSE;

	(*ModeGpa.MODE_WORK_Ring*)10:
		resetAndDisable(alg:=algoritms.Apusk);
		resetAndDisable(alg:=algoritms.SemiAutoPusk);
		resetAndDisable(alg:=algoritms.puskV);
		resetAndDisable(alg:=algoritms.puskK);
		resetAndDisable(alg:=algoritms.testdPmg);
		resetAndDisable(alg:=algoritms.testPms);
		resetAndDisable(alg:=algoritms.ppu);
		algoritms.no.inCanRun:=TRUE;
                    algoritms.no.inOpcCommandsDisabled:=FALSE;
		algoritms.ao.inCanRun:=TRUE;
                    algoritms.ao.inOpcCommandsDisabled:=FALSE;

	(*ModeGpa.MODE_WORK_Line*)11:
		resetAndDisable(alg:=algoritms.Apusk);
		resetAndDisable(alg:=algoritms.SemiAutoPusk);
		resetAndDisable(alg:=algoritms.puskV);
		resetAndDisable(alg:=algoritms.puskK);
		resetAndDisable(alg:=algoritms.testdPmg);
		resetAndDisable(alg:=algoritms.testPms);
		resetAndDisable(alg:=algoritms.ppu);
		resetAndDisable(alg:=algoritms.testIm	 );
		algoritms.no.inCanRun:=TRUE;
                    algoritms.no.inOpcCommandsDisabled:=FALSE;
		algoritms.ao.inCanRun:=TRUE;
                    algoritms.ao.inOpcCommandsDisabled:=FALSE;

	(*ModeGpa.MODE_STOP*)2:
		algoritms.ppu.inCanRun:=TRUE;
                    runIfNotRunning(alg:=algoritms.ppu);
		algoritms.no.inCanRun:=TRUE;
                    algoritms.no.inOpcCommandsDisabled:=FALSE;
		algoritms.ao.inCanRun:=TRUE;
                    algoritms.ao.inOpcCommandsDisabled:=FALSE;
                    (*UnBlockAllProtections(protections);*)
		BlockAllIM(IM);
		algoritms.Remont.inCanRun:=TRUE;
		algoritms.Remont.inOpcCommandsDisabled:=FALSE;
		algoritms.testim.inCanRun:=TRUE;
		algoritms.testim.inOpcCommandsDisabled:=FALSE;
		algoritms.TestProtection.inCanRun:=TRUE;
		algoritms.TestProtection.inOpcCommandsDisabled:=FALSE;
                    algoritms.VibegPNS.inCanRun:=FALSE;
                    algoritms.AutoAvom.inCanRun:=FALSE;
		(*resetAndDisable(alg:=algoritms.puskV);
		resetAndDisable(alg:=algoritms.puskK);
		resetAndDisable(alg:=algoritms.testdPmg);
		resetAndDisable(alg:=algoritms.testPms);*)
	(*ModeGpa.MODE_READY*)3:
		resetAndDisable(alg:=algoritms.Remont);
		resetAndDisable(alg:=algoritms.testim);
		resetAndDisable(alg:=algoritms.TestProtection);
                    algoritms.Apusk.inCanRun:=TRUE;
                    algoritms.Apusk.inOpcCommandsDisabled:=FALSE;
		algoritms.SemiAutoPusk.inCanRun:=TRUE;
                    algoritms.SemiAutoPusk.inOpcCommandsDisabled:=FALSE;
	END_CASE;
END_IF;

(* ---- fb_AnalogParametr.st ---- *)
FUNCTION_BLOCK fb_AnalogParametr

VAR_IN_OUT
	StrAP : struct_AnalogParametr;
END_VAR

VAR
	_sunpackerCommand : fb_sunpackerCommand;
	source : BYTE;
	cmd : BYTE;
	source_for_Status : BYTE;
	cmd_for_Status : BYTE;
	command_error_for_Status : BYTE;
	resetCmdTimer : TON;
	resetCmdTimerPriznak : BOOL;
	secondTact : BOOL;
	inp : LREAL;
	rABS : LREAL;
END_VAR

IF NOT secondTact THEN
	StrAP.Value := StrAP.currentValue;
	secondTact := true;
END_IF;

StrAP.OpcCommandsDisabled := StrAP.inOpcCommandsDisabled;

 (* ---- Если управление с ВУ заблокировано, то передаем команду из алгоритма ---- *)
IF StrAP.inOpcCommandsDisabled THEN
	StrAP.inCommand := StrAP.inCommand_Alg;
ELSE (* иначе передаем команду с АРМа*)
	StrAP.inCommand := StrAP.inCommand_ARM;
END_IF;

_sunpackerCommand(command := StrAP.inCommand);
	source := _sunpackerCommand.source;
	cmd := _sunpackerCommand.cmd;

IF cmd <> 0 AND StrAP.newValue <> StrAP.Value and (((NOT StrAP.opcCommandsDisabled) AND source > 0) OR source = 0) then
	CASE BYTE_TO_INT(cmd) OF
	(*cmd_ChangeValue*) 1 :
				StrAP.isValidValue := TRUE;
				IF StrAP.minVal_ISVALIDREF AND StrAP.isValidValue THEN
					IF StrAP.newValue < StrAP.minVal THEN
						StrAP.isValidValue := FALSE;
					END_IF;
				END_IF;
				IF StrAP.maxVal_ISVALIDREF AND StrAP.isValidValue THEN
					IF StrAP.newValue > StrAP.maxVal THEN
						StrAP.isValidValue := FALSE;
					END_IF;
				END_IF;
				IF StrAP.maxStep_ISVALIDREF AND StrAP.isValidValue  THEN
					inp := StrAP.Value - StrAP.newValue;
					IF inp < 0.0 THEN
						rABS := -inp;
					ELSE
						rABS := inp;
					END_IF;
					IF rABS > StrAP.maxStep THEN
						StrAP.isValidValue := FALSE;
					END_IF;
				END_IF;
				IF StrAP.isValidValue THEN
					StrAP.Value := StrAP.newValue;
					command_error_for_Status := 0;
				ELSE
					command_error_for_Status := cmd;
				END_IF;
	END_CASE;
	source_for_Status := source;
	cmd_for_Status := cmd;
	resetCmdTimer(IN := FALSE);
	resetCmdTimerPriznak := TRUE;
END_IF;

resetCmdTimer(IN := resetCmdTimerPriznak, PT := T#5S);
IF resetCmdTimer.Q THEN
	resetCmdTimerPriznak := FALSE;
	source_for_Status := 0;
	cmd_for_Status := 0;
	command_error_for_Status := 0;
END_IF;

StrAP.status := SHL(BYTE_TO_DWORD(source_for_Status), 29)
			OR SHL(BYTE_TO_DWORD(cmd_for_Status), 26)
			OR SHL(BYTE_TO_DWORD(command_error_for_Status), 23)
			OR SHL(BOOL_TO_DWORD(StrAP.OpcCommandsDisabled ), 21);

(* ---- fb_AnalogParametr_Init.st ---- *)
FUNCTION_BLOCK fb_AnalogParametr_Init

VAR_INPUT
	data_Ini : BOOL; (*Флаг необходимости инициализации параметров.*)
	currentValue : LREAL;
	minVal : LREAL;
	maxVal : LREAL;
	maxStep : LREAL;
	minVal_ISVALIDREF : BOOL;
	maxVal_ISVALIDREF : BOOL;
	maxStep_ISVALIDREF : BOOL;
END_VAR

VAR_IN_OUT
	strAP : struct_AnalogParametr;
END_VAR

VAR_OUTPUT
	Init : BOOL          := FALSE; (*Флаг успешно выполненной инициализации.*)
END_VAR

(*****            Функциональный блок переинициализации Аналогового параметра.            *****)
     Init := false;

    IF data_Ini THEN                            (* Параметрам требуется переинициализация. *)
        strAP.currentValue          := currentValue;
        strAP.minVal                := minVal;
        strAP.maxVal                := maxVal;
        strAP.maxStep               := maxStep;
        strAP.minVal_ISVALIDREF     := minVal_ISVALIDREF;
        strAP.maxVal_ISVALIDREF     := maxVal_ISVALIDREF;
        strAP.maxStep_ISVALIDREF    := maxStep_ISVALIDREF;

        data_Ini:=false;
        Init := TRUE;
     END_IF;
     IF Init THEN
        currentValue:= 0.0;
        minVal:= 0.0;
        maxVal:= 0.0;
        maxStep:= 0.0;
        minVal_ISVALIDREF:= false;
        maxVal_ISVALIDREF:= false;
        maxStep_ISVALIDREF:= false;
     END_IF;

(* ---- fb_AntiPompagAlg.st ---- *)
FUNCTION_BLOCK fb_AntiPompagAlg

VAR
	tableQ_min : fb_TableValue_Min;
	tableQ_max : fb_TableValue_Max;
	fb_Rashod : fb_RashodAlg;
	fb_Zapas : fb_ZapasAlg;
END_VAR

VAR_IN_OUT
	Kran6 : struct_Kran;
	StrAlg : struct_Alg;
	Rashod : struct_AI;
	Zapas : struct_AI;
END_VAR

VAR_INPUT
	P_gasIn : struct_AI;
	T_gasIn : struct_AI;
	dP_konf : struct_AI;
	UgolVNA : struct_AnalogParametr;
	K : struct_AnalogParametr;
	A : struct_AnalogParametr;
	y0 : struct_AnalogParametr;
END_VAR

VAR
	Q_max : LREAL;
	Q_min : LREAL;
	pompaj : BOOL;
	_statusAi : TYPE_StatusAi;
	_statusDualInput : TYPE_statusDualInput;
	_sunpackerCommand : fb_sunpackerCommand;
	source : BYTE;
	cmd : BYTE;
	lastCmd : BYTE;
	source_for_Status : BYTE;
	cmd_for_Status : BYTE;
	command_error_for_Status : BYTE;
	resetCmdTimer : TON;
	resetCmdTimerPriznak : BOOL;
END_VAR

tableQ_min(parametr:=LREAL_TO_REAL(UgolVNA.Value));

tableQ_max(parametr:=LREAL_TO_REAL(UgolVNA.Value));

Q_min:=REAL_TO_LREAL(tableQ_min.actualValue);

Q_max:=REAL_TO_LREAL(tableQ_max.actualValue);

fb_Rashod(StrAi:=Rashod, P_gasIn:=P_gasIn, T_gasIn:=T_gasIn, dP_konf:=dP_konf, K:=K, A:=A, y0:=y0);

fb_Zapas(StrAi:=Zapas, Q_actual:=Rashod, Q_min:=Q_min, Q_max:=Q_max);

StrAlg.CanRun := StrAlg.inCanRun;

StrAlg.OpcCommandsDisabled := StrAlg.inOpcCommandsDisabled;

IF StrAlg.isRuning THEN

StrAlg.hasError := (Rashod.interval < _statusAi.normal);

pompaj:= (Rashod.interval>=_statusAi.normal) AND (Rashod.value <= Q_min);

IF pompaj THEN
          Kran6.inOpcCommandsDisabled:=TRUE;
	Kran6.inCommand_Alg := 1;  (*cmd_open*)
END_IF;

StrAlg.isEnded := Kran6.onStatus = _statusDualInput.STATUS_ON ;

END_IF;

(* ---- Если управление с ВУ заблокировано, то передаем команду из алгоритма ---- *)
IF StrAlg.inOpcCommandsDisabled THEN
	StrAlg.inCommand := StrAlg.inCommand_Alg;
ELSE (* иначе передаем команду с АРМа*)
	StrAlg.inCommand := StrAlg.inCommand_ARM;
END_IF;

_sunpackerCommand(command := StrAlg.inCommand);
	source := _sunpackerCommand.source;
	cmd := _sunpackerCommand.cmd;

IF cmd <> 0 AND lastCmd <> cmd AND (((NOT StrAlg.opcCommandsDisabled) AND source > 0) OR source = 0) then
	CASE BYTE_TO_INT(cmd) OF
		(*cmdRun*) 1: 	IF (StrAlg.CanRun) THEN
					StrAlg.isRuning := TRUE;
					StrAlg.isEnded := FALSE;
					StrAlg.hasError 	:= FALSE;

                                                  (*****************       OnRun       *****************)

					cmd_for_Status := cmd;
					source_for_Status := source;
					command_error_for_Status := 0;
				ELSE
					StrAlg.isRuning := FALSE;
					StrAlg.isEnded := FALSE;
					StrAlg.hasError 	:= FALSE;

					cmd_for_Status := 0;
					source_for_Status := source;
					command_error_for_Status := cmd;
				END_IF;
		(*cmdReset*) 2: 	StrAlg.isRuning := FALSE;
				StrAlg.isEnded := FALSE;
				StrAlg.hasError 	:= FALSE;
                                        (*****************       OnReset       *****************)

                                                  pompaj:= FALSE;
                                                  Kran6.inOpcCommandsDisabled:=FALSE;
				cmd_for_Status := cmd;
				source_for_Status := source;
				command_error_for_Status := 0;
	END_CASE;
	resetCmdTimer(IN := false);
	resetCmdTimerPriznak := TRUE;
END_IF;
lastCmd := cmd;

resetCmdTimer(IN := resetCmdTimerPriznak, PT := T#5S);
IF resetCmdTimer.Q THEN
	resetCmdTimerPriznak := FALSE;
	source_for_Status := 0;
	cmd_for_Status := 0;
	command_error_for_Status := 0;
END_IF;

StrAlg.status :=  SHL(BYTE_TO_DWORD(source_for_Status), 29)
			OR SHL(BYTE_TO_DWORD(cmd_for_Status), 26)
			OR SHL(BYTE_TO_DWORD(command_error_for_Status), 23)
			OR SHL(BOOL_TO_DWORD(StrAlg.OpcCommandsDisabled ), 21)
			OR SHL(BOOL_TO_DWORD(StrAlg.hasError),4)
			OR SHL(BOOL_TO_DWORD(StrAlg.CanRun),2)
			OR SHL(BOOL_TO_DWORD(StrAlg.isEnded),1)
			OR BOOL_TO_DWORD(StrAlg.isRuning);

(* ---- fb_AO_Init.st ---- *)
FUNCTION_BLOCK fb_AO_Init

VAR_INPUT
	data_Ini : BOOL; (*Флаг необходимости инициализации параметров.*)
	outLL : LREAL          := 4000.0;
	outHL : LREAL          := 20000.0;
	newLL : LREAL;
	newHL : LREAL;
	newLL_ISVALIDREF : BOOL;
	newHL_ISVALIDREF : BOOL;
END_VAR

VAR_IN_OUT
	strAO : struct_AO; (*Дескриптор AI-канала.*)
END_VAR

VAR_OUTPUT
	Init : BOOL          := FALSE; (*Флаг успешно выполненной инициализации.*)
END_VAR

(*****            Функциональный блок переинициализации структуры-дескриптора канала аналогового ввода.            *****)

 Init := FALSE;

    IF data_Ini THEN                            (* Параметрам требуется переинициализация. *)
        strAO.outLL                := outLL;
        strAO.outHL                := outHL;
        strAO.newLL                := newLL;
        strAO.newHL                := newHL;
        strAO.newLL_ISVALIDREF     := newLL_ISVALIDREF;
        strAO.newHL_ISVALIDREF     := newHL_ISVALIDREF;
        data_Ini:=FALSE;
        Init := TRUE;
    END_IF;
 IF Init THEN
       (* outLL:=0.0;*)
       (* outHL:=0.0;*)
        newLL:=0.0;
        newHL:=0.0;
        newLL_ISVALIDREF:= FALSE;
        newHL_ISVALIDREF:= FALSE;
 END_IF;

(* ---- fb_AOSourceMlp.st ---- *)
FUNCTION_BLOCK fb_AOSourceMlp

VAR_IN_OUT
	OutCurrent : TDoubleData; (*Данные для модуля AO.*)
	strAO : struct_AO; (*Текущие параметры канала AO*)
END_VAR

VAR
	_sunpackerCommand : fb_sunpackerCommand;
	source : BYTE;
	source_for_Status : BYTE;
	cmd : BYTE;
	cmd_for_Status : BYTE;
	lastCmd : BYTE;
	command_error_for_Status : BYTE;
	resetCmdTimer : TON;
	resetCmdTimerPriznak : BOOL;
	secondTack : BOOL;
	inOpcCommandsDisabled : BOOL;
END_VAR

VAR_INPUT RETAIN
	retainLL : LREAL;
	retainHL : LREAL;
END_VAR

IF NOT secondTack THEN
          IF (strAO.newLL <> retainLL) AND (retainLL <> 0.0) THEN  strAO.LL := retainLL;
          ELSE strAO.LL:= strAO.newLL; END_IF;
	IF (strAO.newHL <> retainHL) AND (retainHL <> 0.0) THEN  strAO.HL := retainHL;
          ELSE strAO.HL:= strAO.newHL; END_IF;

	secondTack  := FALSE;
END_IF;
strAO.blConnect :=(UINT_TO_WORD(OutCurrent.wFlags) AND 16#0040) <> 0;
strAO.OpcCommandsDisabled := inOpcCommandsDisabled;

_sunpackerCommand(command := strAO.inCommand);
	source := _sunpackerCommand.source;
	cmd := _sunpackerCommand.cmd;

IF cmd <> 0 AND lastCmd <> cmd and (((NOT strAO.opcCommandsDisabled) AND source > 0) OR source = 0) then
	CASE BYTE_TO_INT(cmd) OF
	(*cmd_ChangeValue*) 1 : 	IF ((NOT strAO.newLL_ISVALIDREF) OR (strAO.nValue >= strAO.LL)) AND
                                           ((NOT strAO.newHL_ISVALIDREF) OR (strAO.nValue <= strAO.HL) ) THEN
					strAO.Value := strAO.nValue;
				END_IF;
	(*cmd_ChangeLimits*) 2 : 	strAO.LL := strAO.newLL; retainLL:= strAO.LL;
				strAO.HL := strAO.newHL; retainHL:= strAO.HL;
	END_CASE;
	source_for_Status := source;
	cmd_for_Status := cmd;
	command_error_for_Status := 0;
	resetCmdTimer(IN := FALSE);
	resetCmdTimerPriznak := TRUE;
END_IF;
lastCmd := cmd;

IF (strAO.HL <> strAO.LL) THEN
	OutCurrent.dblValue := ((strAO.Value - strAO.LL) * (strAO.outHL-strAO.outLL)/(strAO.HL - strAO.LL )) + strAO.outLL;
END_IF;

resetCmdTimer(IN := resetCmdTimerPriznak, PT := T#5S);
IF resetCmdTimer.Q THEN
	resetCmdTimerPriznak := FALSE;
	source_for_Status := 0;
	cmd_for_Status := 0;
	command_error_for_Status := 0;
END_IF;

strAO.status := SHL(BYTE_TO_DWORD(source_for_Status), 29)
			OR SHL(BYTE_TO_DWORD(cmd_for_Status), 26)
			OR SHL(BYTE_TO_DWORD(command_error_for_Status), 23)
			OR SHL(BOOL_TO_DWORD(strAO.OpcCommandsDisabled ), 21);

(* ---- fb_AutoAvomAlg.st ---- *)
FUNCTION_BLOCK fb_AutoAvomAlg

VAR_IN_OUT
	StrAlg : struct_Alg;
	im1 : struct_Switch;
	im2 : struct_Switch;
END_VAR

VAR_INPUT
	ai : struct_AI;
END_VAR

VAR_IN_OUT
	on1Temperature : struct_AnalogParametr;
	on2Temperature : struct_AnalogParametr;
	hystereses : struct_AnalogParametr;
END_VAR

VAR
	_sunpackerCommand : fb_sunpackerCommand;
	_statusAi : TYPE_StatusAi;
	_statusDualInput : TYPE_statusDualInput;
	_commandDualInput : TYPE_commandDualInput;
	source : BYTE;
	cmd : BYTE;
	lastCmd : BYTE;
	source_for_Status : BYTE;
	cmd_for_Status : BYTE;
	command_error_for_Status : BYTE;
	resetCmdTimer : TON;
	resetCmdTimerPriznak : BOOL;
	onInit : BOOL;
END_VAR

(*
IF NOT onInit THEN
StrAlg.inCanRun:=TRUE;
onInit:=TRUE;
END_IF;
*)

IF StrAlg.isRuning THEN

StrAlg.hasError := im1.CommandFault OR im2.CommandFault OR (ai.interval<_statusAi.normal);

    IF (ai.interval>=_statusAi.normal) THEN

          IF (ai.value>= on1Temperature.Value) THEN
              IF im1.onStatus <> _statusDualInput.STATUS_ON THEN
	       im1.inCommand_Alg:=BYTE_TO_WORD(_commandDualInput.CMD_ON); (*cmd_on*)
              END_IF;
          END_IF;

          IF  ai.value < (on1Temperature.Value - hystereses.Value) THEN
              IF im1.onStatus <> _statusDualInput.STATUS_OFF THEN
	       im1.inCommand_Alg:=BYTE_TO_WORD(_commandDualInput.CMD_OFF);
              END_IF;
          END_IF;

           IF (ai.value>= on2Temperature.Value) THEN
              IF im2.onStatus <> _statusDualInput.STATUS_ON THEN
	       im2.inCommand_Alg:=BYTE_TO_WORD(_commandDualInput.CMD_ON); (*cmd_on*)
              END_IF;
          END_IF;

          IF  ai.value < (on2Temperature.Value - hystereses.Value) THEN
              IF im2.onStatus <> _statusDualInput.STATUS_OFF THEN
	       im2.inCommand_Alg:=BYTE_TO_WORD(_commandDualInput.CMD_OFF);
              END_IF;
          END_IF;
     END_IF;

END_IF;

StrAlg.CanRun := StrAlg.inCanRun;

StrAlg.OpcCommandsDisabled := StrAlg.inOpcCommandsDisabled;

(* ---- Если управление с ВУ заблокировано, то  передаем команду из алгоритма ---- *)
IF StrAlg.inOpcCommandsDisabled THEN
	StrAlg.inCommand := StrAlg.inCommand_Alg;
ELSE (* иначе передаем команду с АРМа*)
	StrAlg.inCommand := StrAlg.inCommand_ARM;
END_IF;

_sunpackerCommand(command := StrAlg.inCommand);
	source := _sunpackerCommand.source;
	cmd := _sunpackerCommand.cmd;

IF cmd <> 0 AND lastCmd <> cmd AND (((NOT StrAlg.opcCommandsDisabled) AND source > 0) OR source = 0) then
	CASE BYTE_TO_INT(cmd) OF
		(*cmdRun*) 1: 	IF (StrAlg.CanRun) THEN
					StrAlg.isRuning := TRUE;
					StrAlg.isEnded := FALSE;
					StrAlg.hasError := FALSE;
                                                  StrAlg.inOpcCommandsDisabled:=FALSE;
					im1.inOpcCommandsDisabled:=TRUE;
                                                  im2.inOpcCommandsDisabled:=TRUE;
					cmd_for_Status := cmd;
					source_for_Status := source;
					command_error_for_Status := 0;
				ELSE
					StrAlg.isRuning := FALSE;
					StrAlg.isEnded := FALSE;
					StrAlg.hasError 	:= FALSE;

					cmd_for_Status := 0;
					source_for_Status := source;
					command_error_for_Status := cmd;
				END_IF;
		(*cmdReset*) 2: 	StrAlg.isRuning := FALSE;
				StrAlg.isEnded := FALSE;
				StrAlg.hasError 	:= FALSE;
                                        StrAlg.inOpcCommandsDisabled:=FALSE;
                                        im1.inOpcCommandsDisabled:=FALSE;
                                        im2.inOpcCommandsDisabled:=FALSE;
                                        im1.inCommand_Alg:=0;
                                        im2.inCommand_Alg:=0;
				cmd_for_Status := cmd;
				source_for_Status := source;
				command_error_for_Status := 0;
	END_CASE;
	resetCmdTimer(IN := false);
	resetCmdTimerPriznak := TRUE;
END_IF;
lastCmd := cmd;

resetCmdTimer(IN := resetCmdTimerPriznak, PT := T#5S);
IF resetCmdTimer.Q THEN
	resetCmdTimerPriznak := FALSE;
	source_for_Status := 0;
	cmd_for_Status := 0;
	command_error_for_Status := 0;
END_IF;

(*TODO: TYPE PROGRAM CODE HERE*)
StrAlg.status :=  SHL(BYTE_TO_DWORD(source_for_Status), 29)
			OR SHL(BYTE_TO_DWORD(cmd_for_Status), 26)
			OR SHL(BYTE_TO_DWORD(command_error_for_Status), 23)
			OR SHL(BOOL_TO_DWORD(StrAlg.OpcCommandsDisabled ), 21)
			OR SHL(BOOL_TO_DWORD(StrAlg.hasError),4)
			OR SHL(BOOL_TO_DWORD(StrAlg.CanRun),2)
			OR SHL(BOOL_TO_DWORD(StrAlg.isEnded),1)
			OR BOOL_TO_DWORD(StrAlg.isRuning);

(* ---- fb_AutoNUAlg.st ---- *)
FUNCTION_BLOCK fb_AutoNUAlg

VAR_IN_OUT
	StrAlg : struct_Alg;
	nu1 : struct_OilPump;
	nu2 : struct_OilPump;
END_VAR

VAR_INPUT
	dPoil : struct_AI;
END_VAR

VAR_IN_OUT
	mainNU : struct_DiscretParametr;
	Lowdp_di : struct_singleSignal;
	Ust_Swap : struct_AnalogParametr;
END_VAR

VAR
	_prevMainNU : UINT;
	_sunpackerCommand : fb_sunpackerCommand;
	_statusAi : TYPE_StatusAi;
	_statusDualInput : TYPE_statusDualInput;
	_commandDualInput : TYPE_commandDualInput;
	source : BYTE;
	cmd : BYTE;
	lastCmd : BYTE;
	source_for_Status : BYTE;
	cmd_for_Status : BYTE;
	command_error_for_Status : BYTE;
	resetCmdTimer : TON;
	waitPressure : TON;
	waitPressureTrig : R_TRIG;
	resetCmdTimerPriznak : BOOL;
	onInit : BOOL;
	onStart : BOOL;
END_VAR

VAR_EXTERNAL
	NotHasRezervNU : BOOL;
	Reset_HasNU : BOOL;
END_VAR

IF NOT onInit THEN
StrAlg.inCanRun:=TRUE;
StrAlg.inOpcCommandsDisabled:=TRUE;
(*nu1.Osnovnoy:=TRUE; nu2.Osnovnoy:=FALSE;*)
onInit:=TRUE;
END_IF;

IF Reset_HasNU THEN
nu1.inBlocked:=FALSE;
nu2.inBlocked:=FALSE;
END_IF;

NotHasRezervNU:=(nu1.Blocked OR nu2.Blocked);

IF StrAlg.isRuning THEN

StrAlg.hasError := nu1.CommandFault OR nu2.CommandFault OR (dPoil.interval<_statusAi.normal);

 IF mainNU.value<>_prevMainNU OR NOT onStart THEN

        CASE mainNU.value OF
	0: nu1.Osnovnoy:=TRUE; nu2.Osnovnoy:=FALSE;
	1: nu1.Osnovnoy:=FALSE; nu2.Osnovnoy:=TRUE;

        END_CASE;

    IF  nu1.Osnovnoy AND NOT nu1.Blocked THEN
        nu1.inCommand_Alg:=BYTE_TO_WORD(_commandDualInput.CMD_ON);
    ELSIF NOT NotHasRezervNU THEN
        nu1.inCommand_Alg:=BYTE_TO_WORD(_commandDualInput.CMD_OFF);
    END_IF;

    IF  nu2.Osnovnoy AND NOT nu2.Blocked THEN
        nu2.inCommand_Alg:=BYTE_TO_WORD(_commandDualInput.CMD_ON);
     ELSIF NOT NotHasRezervNU THEN
        nu2.inCommand_Alg:=BYTE_TO_WORD(_commandDualInput.CMD_OFF);
    END_IF;
      onStart:=TRUE;
     _prevMainNU:=mainNU.value;
 END_IF;

  (*IF (nu1.onStatus = _statusDualInput.STATUS_On) OR (nu2.onStatus = _statusDualInput.STATUS_On) THEN*)
    (*Если через 5С насос не нагнал 100кПа масла - он сломался и надо переключить насос*)
    IF dPoil.interval>= _statusAi.NORMAL THEN
          waitPressure(IN:=(dPoil.value<Ust_Swap.Value OR LowdP_DI.q) AND NOT NotHasRezervNU, PT:= T#5S);
    ELSE
	waitPressure(IN:=(FALSE));
    END_IF;

    waitPressureTrig(CLK:=waitPressure.Q);
    IF waitPressureTrig.Q THEN
	(*IF nu1.onStatus = _statusDualInput.STATUS_ON THEN*)
           IF mainNU.value = 0 THEN
		nu1.inBlocked:=TRUE;
                    nu1.inCommand_Alg:=BYTE_TO_WORD(_commandDualInput.CMD_OFF);
			(*IF 	mainNU.value = 0 THEN*)
                                        setValue(mainNU, 1);
			(*END_IF;*)
	END_IF;

	(*IF nu2.onStatus = _statusDualInput.STATUS_ON THEN*)
          IF mainNU.value = 1 THEN
		nu2.inBlocked:=TRUE;
                    nu2.inCommand_Alg:=BYTE_TO_WORD(_commandDualInput.CMD_OFF);
			(*IF 	mainNU.value = 1 THEN*)
				setValue(mainNU, 0);
			(*END_IF;*)
	END_IF;
    END_IF;
 (* END_IF;*)

END_IF;

StrAlg.CanRun := StrAlg.inCanRun;

StrAlg.OpcCommandsDisabled := StrAlg.inOpcCommandsDisabled;

(* ---- Если управление с ВУ заблокировано, то  передаем команду из алгоритма ---- *)
IF StrAlg.inOpcCommandsDisabled THEN
	StrAlg.inCommand := StrAlg.inCommand_Alg;
ELSE (* иначе передаем команду с АРМа*)
	StrAlg.inCommand := StrAlg.inCommand_ARM;
END_IF;

_sunpackerCommand(command := StrAlg.inCommand);
	source := _sunpackerCommand.source;
	cmd := _sunpackerCommand.cmd;

IF cmd <> 0 AND lastCmd <> cmd AND (((NOT StrAlg.opcCommandsDisabled) AND source > 0) OR source = 0) then
	CASE BYTE_TO_INT(cmd) OF
		(*cmdRun*) 1: 	IF (StrAlg.CanRun) THEN
					StrAlg.isRuning := TRUE;
					StrAlg.isEnded := FALSE;
					StrAlg.hasError := FALSE;

                                                  (*****************       OnRun       *****************)
					nu1.inOpcCommandsDisabled:=TRUE;
                                                  nu2.inOpcCommandsDisabled:=TRUE;

					cmd_for_Status := cmd;
					source_for_Status := source;
					command_error_for_Status := 0;
				ELSE
					StrAlg.isRuning := FALSE;
					StrAlg.isEnded := FALSE;
					StrAlg.hasError 	:= FALSE;

					cmd_for_Status := 0;
					source_for_Status := source;
					command_error_for_Status := cmd;
				END_IF;
		(*cmdReset*) 2: 	StrAlg.isRuning := FALSE;
				StrAlg.isEnded := FALSE;
				StrAlg.hasError 	:= FALSE;

                                        (*****************       OnReset       *****************)
                                        waitPressure(IN:=(FALSE));
                                        onStart:=FALSE;

				cmd_for_Status := cmd;
				source_for_Status := source;
				command_error_for_Status := 0;
	END_CASE;
	resetCmdTimer(IN := false);
	resetCmdTimerPriznak := TRUE;
END_IF;
lastCmd := cmd;

resetCmdTimer(IN := resetCmdTimerPriznak, PT := T#5S);
IF resetCmdTimer.Q THEN
	resetCmdTimerPriznak := FALSE;
	source_for_Status := 0;
	cmd_for_Status := 0;
	command_error_for_Status := 0;
END_IF;

(*TODO: TYPE PROGRAM CODE HERE*)
StrAlg.status :=  SHL(BYTE_TO_DWORD(source_for_Status), 29)
			OR SHL(BYTE_TO_DWORD(cmd_for_Status), 26)
			OR SHL(BYTE_TO_DWORD(command_error_for_Status), 23)
			OR SHL(BOOL_TO_DWORD(StrAlg.OpcCommandsDisabled ), 21)
                              OR SHL(BOOL_TO_DWORD(NotHasRezervNU), 15)
			OR SHL(BOOL_TO_DWORD(StrAlg.hasError),4)
			OR SHL(BOOL_TO_DWORD(StrAlg.CanRun),2)
			OR SHL(BOOL_TO_DWORD(StrAlg.isEnded),1)
			OR BOOL_TO_DWORD(StrAlg.isRuning);

(* ---- fb_AutoPnsAlg.st ---- *)
FUNCTION_BLOCK fb_AutoPnsAlg

VAR_IN_OUT
	StrAlg : struct_Alg;
	Nasos : struct_Switch;
END_VAR

VAR_INPUT
	diPlow : struct_singleSignal;
	Poil : struct_AI;
	Ust_Run : struct_AnalogParametr;
	Ust_Stop : struct_AnalogParametr;
END_VAR

VAR
	_sunpackerCommand : fb_sunpackerCommand;
	_statusAi : TYPE_StatusAi;
	_statusDualInput : TYPE_statusDualInput;
	_commandDualInput : TYPE_commandDualInput;
	source : BYTE;
	cmd : BYTE;
	lastCmd : BYTE;
	source_for_Status : BYTE;
	cmd_for_Status : BYTE;
	command_error_for_Status : BYTE;
	resetCmdTimer : TON;
	resetCmdTimerPriznak : BOOL;
	onInit : BOOL;
	onTrig : R_TRIG;
	offTrig : R_TRIG;
	waitOn : TON;
	waitOff : TON;
END_VAR

VAR_EXTERNAL
	AlgTimers : struct_AlgTimers;
END_VAR

IF NOT onInit THEN
StrAlg.inOpcCommandsDisabled:=TRUE;
StrAlg.inCanRun:=TRUE;
onInit:=TRUE;
END_IF;

IF StrAlg.isRuning THEN

StrAlg.hasError := Nasos.CommandFault OR (Poil.interval < _statusAi.normal OR NOT diPlow.reliability);

    IF (Poil.Interval >= _statusAi.normal) THEN
    waitOn(IN:=Poil.Value <= Ust_Run.value OR diPlow.q, PT := T#1S);
    waitOff(IN:= Poil.Value >= Ust_Stop.value, PT := T#300S);

    ELSE
    waitOn(IN:=diPlow.Q, PT := T#1S);
    END_IF;

onTrig(CLK:=waitOn.Q);
offTrig(CLK:=waitOff.Q);
    IF (Poil.Value>=Ust_Stop.value) AND Nasos.inopcCommandsDisabled THEN
        Nasos.inopcCommandsDisabled:=FALSE;
    END_IF;

    IF onTrig.Q THEN
    Nasos.inopcCommandsDisabled:=TRUE;
    Nasos.inCommand_Alg:=BYTE_TO_WORD(_commandDualInput.CMD_ON);
    END_IF;

    IF offTrig.Q THEN
        IF NOT (Nasos.onStatus=_statusDualInput.STATUS_OFF) THEN
        Nasos.inopcCommandsDisabled:=TRUE;
        Nasos.inCommand_Alg:=BYTE_TO_WORD(_commandDualInput.CMD_OFF);
        END_IF;
    END_IF;

AlgTimers.AutoPns_OnTimer:=UDINT_TO_UINT(TIME_TO_UDINT(waitOn.PT - waitOn.ET)/1000);
AlgTimers.AutoPns_OffTimer:=UDINT_TO_UINT(TIME_TO_UDINT(waitOff.PT -waitOff.ET)/1000);

END_IF;

StrAlg.CanRun := StrAlg.inCanRun;

StrAlg.OpcCommandsDisabled := StrAlg.inOpcCommandsDisabled;
